// TIA Portal project "plc-programs_V19_S7-1500_PLCSIM_advanced" (V19)
// Vorlageprojekt für das Buch mit Zielsystem S7-1200

(* hardware
DEVICE "S7-1500/ET200MP station_1"  S7-1500 station
   slot 0: "Rail_0"  Rack  6ES7 590-1***0-0AA0
   slot 1: "PLC_1"  CPU 1511-1 PN  6ES7 511-1AK01-0AB0  V2.9
      slot 3: "CPU display_1"  6ES7591-1AA00-0AA0
      slot 32768: "PROFINET interface_1"  X1
         slot 32769: "Port_1"  X1 P1
         slot 32770: "Port_2"  X1 P2
      slot 34817: "Virtual CP interface port_1"  Virtual CP interface port  Virtual CP interface port
*)

// ===== PLC "PLC_1"  CPU 1511-1 PN =====

VAR_GLOBAL   // PLC tag table "Default tag table"
   "Tag_11" AT %M2.4 : Bool;
   "Tag_12" AT %M3.1 : Bool;
END_VAR

VAR_GLOBAL   // PLC tag table "Tag table_Stations123"
   "DI_S1_DiffEntry" AT %I0.2 : Bool;   // S1 item present at infeed
   "DI_S1_VisColor" AT %I0.3 : Bool;   // S1 color/vision detection (blue)
   "DI_S1_PusherBack" AT %I0.4 : Bool;   // S1 pusher fully retracted (home)
   "DI_S1_PusherFront" AT %I0.5 : Bool;   // S1 pusher fully extended
   "DO_S1_Belt2m_A" AT %Q0.1 : Bool;   // S1 short belt A (infeed segment)
   "DO_S2_Belt2m_B" AT %Q0.2 : Bool;   // S2 short belt B (next segment)
   "DO_S1_Belt4m" AT %Q0.3 : Bool;   // S1 long belt past the vision sensor
   "DO_S1_Emitter" AT %Q0.4 : Bool;   // S1 raw material emitter
   "DO_S1_Remover" AT %Q0.5 : Bool;   // S1 rejected blue lid remover
   "DO_S1_Pusher" AT %Q0.6 : Bool;   // S1 pusher extend coil
   "DI_S2_DiffStop0" AT %I0.6 : Bool;   // S2 part present at stop blade 0
   "DI_S2_DiffEntry" AT %I0.7 : Bool;   // S2 part entering station 2
   "r_S2_ArmZpos" AT %ID30 : Real;   // S2 Two-Axis Pick & Place Z axis feedback
   "r_S2_ArmXpos" AT %ID34 : Real;   // S2 Two-Axis Pick & Place X axis feedback
   "DI_S2_ArmRotating" AT %I1.4 : Bool;   // S2 gripper currently rotating
   "DO_S2_Emitter" AT %Q0.7 : Bool;   // S2 base emitter
   "DO_S2_Belt2m_C" AT %Q1.0 : Bool;   // S2 belt carrying parts into the station
   "r_S2_CmdMoveZ" AT %QD30 : Real;   // S2 setpoint for Z axis
   "r_S2_CmdMoveX" AT %QD34 : Real;   // S2 setpoint for X axis
   "DO_S2_Grabe" AT %Q1.2 : Bool;   // S2 gripper close coil
   "DO_S2_RotateRight" AT %Q1.3 : Bool;   // S2 rotate gripper clockwise
   "DO_S2_RotateLeft" AT %Q1.4 : Bool;   // S2 rotate gripper counter-clockwise
   "DO_S2_StopBlade0" AT %Q1.5 : Bool;   // S2 stop blade 0 (near entry)
   "DO_S2_StopBlade1" AT %Q1.6 : Bool;   // S2 stop blade 1 (near assembly)
   "DI_S3_DiffEntry" AT %I1.0 : Bool;   // S3 item entering roller conveyor
   "DI_S3_EntryPart" AT %I1.5 : Bool;   // S3 fingerprint/part present at entry
   "DI_S3_PusherLimit" AT %I1.6 : Bool;   // S3 pusher reached its limit
   "DI_S3_Clamped" AT %I1.7 : Bool;   // S3 clamp closed sensor
   "DI_S3_PalletEntry" AT %I2.0 : Bool;   // S3 empty pallet arrived at loading position
   "DI_S3_PalletLoaded" AT %I2.1 : Bool;   // S3 pallet loaded with a row of items
   "DI_S3_PlateLimit" AT %I2.2 : Bool;   // S3 plate reached its travel limit
   "DI_S3_ElevatorMoving" AT %I2.3 : Bool;   // S3 elevator in motion
   "DO_S3_Clamp" AT %Q2.1 : Bool;   // S3 clamp open/close command
   "DO_S3_OpenPlate" AT %Q2.2 : Bool;   // S3 release plate command
   "DO_S3_PalletLoad" AT %Q2.3 : Bool;   // S3 start loading the pallet
   "DO_S3_Emitter" AT %Q3.2 : Bool;   // S3 Pallet emitter
   "DO_S3_Roller4m_A" AT %Q2.5 : Bool;   // S3 roller conveyor segment A (infeed)
   "DO_S3_Roller4m_B" AT %Q2.6 : Bool;   // S3 roller conveyor segment B (outfeed)
   "DO_S3_ElevatorUp" AT %Q2.7 : Bool;   // S3 raise elevator
   "DO_S3_ElevatorDown" AT %Q3.0 : Bool;   // S3 lower elevator
   "DO_S3_MoveToLimit" AT %Q3.1 : Bool;   // S3 drive elevator to its limit
   "DI_S2_DiffStop1" AT %I1.1 : Bool;   // S2 part present at stop blade 1
   "DI_S2_DiffArmHome" AT %I1.2 : Bool;   // S2 Two-Axis Pick & Place at home
   "DI_S2_ItemDetected" AT %I1.3 : Bool;   // S2 assembly station sees the item
   "DO_S2_Belt2m_D" AT %Q1.1 : Bool;   // S2 outfeed belt after assembly
   "DO_S3_PalletizerBelt" AT %Q1.7 : Bool;   // S3 palletizer transport belt
   "DO_S3_Push" AT %Q2.0 : Bool;   // S3 item pusher (into elevator)
   "DI_S3_PalletExit" AT %I2.4 : Bool;   // S3 finished pallet at exit sensor
   "DO_S3_Remover" AT %Q3.3 : Bool;   // S3 finished-pallet remover
END_VAR

VAR_GLOBAL   // PLC tag table "Tag table_ControlPanel"
   "EStop" AT %I2.5 : Bool;
   "Btn_EstopReset" AT %I2.6 : Bool;
   "Start_Btn" AT %I2.7 : Bool;
   "Stop_Bnt" AT %I3.0 : Bool;
   "AutoMode_S1" AT %I3.1 : Bool;
   "ManualMode_S1" AT %I3.2 : Bool;
   "Lamp_Auto" AT %Q3.4 : Bool;
   "Lamp_Fault" AT %Q3.5 : Bool;
   "Lamp_Run" AT %Q3.6 : Bool;
   "Btn_Start_active" AT %Q3.7 : Bool;
   "Btn_Stop_active" AT %Q4.0 : Bool;
   "EStopReset_Active" AT %Q4.1 : Bool;
   "Btn_ResetCount" AT %I3.3 : Bool;
   "Final_Product_Count" AT %QD38 : DInt;
   "HMI_Start_Btn" AT %M5.0 : Bool;
   "HMI_Sop_Btn" AT %M5.1 : Bool;
   "HMI_CountReset" AT %M5.2 : Bool;
END_VAR

VAR_GLOBAL   // PLC tag table "Tag_table_KPIs"
   "TotalItemsRejected" AT %QD42 : DInt;   // Total rejected items (from FC2 quality reject)
   "TotalRunTime" AT %QD46 : DInt;   // Total run time in seconds
   "ShiftPlannedTime" AT %MW50 : Int;   // Planned production time in seconds (e.g. 28800 = 8h)
   "IdealRate" AT %QD52 : Real;   // Ideal rate items/sec (e.g. 2.5)
   "ActiveAlarmCount" AT %QW56 : Int;   // Number of active alarms
   "TotalDowntime" AT %QD58 : DInt;   // Total downtime in seconds
   "RejectPulse" AT %M2.0 : Bool;   // One-shot pulse on each reject event
   "ProductionPulse" AT %M2.1 : Bool;   // One-shot pulse on each produced item
   "RunTimeEnable" AT %M2.2 : Bool;   // TRUE while line is running (for TON)
   "DowntimeEnable" AT %M2.3 : Bool;   // TRUE while line is stopped (for TON)
   "LidsCount" AT %MD20 : DInt;
   "Alarm_EStop" AT %M4.0 : Bool;
   "Alarm_Fault" AT %M4.1 : Bool;
   "Alarm_LowProduction" AT %M4.2 : Bool;
   "Alarm_HighSort" AT %M4.3 : Bool;
   "Alarm_S2_GripperFault" AT %M4.4 : Bool;
END_VAR

VAR_GLOBAL   // PLC tag table "Standard-Variablentabelle"
   "Tag_1" AT %Q0.0 : Bool;   // Indicates initial communication setup cycle is complete
   "Tag_2" AT %I0.0 : Bool;   // Factory I/O communication link health bit
   "Tag_3" AT %I0.1 : Bool;   // Controls data driver execution for Factory I/O I/O mapping
   "b_S1_PusherReq" AT %M0.0 : Bool;   // S1 pusher request latch
   "Cnt_S3_ItemsInRow" AT %MW20 : Int;   // S3 count of items in current row (CTU counter_0 CV)
   "b_S3_Trig_ElevatorStop" AT %M0.2 : Bool;   // N_TRIG on ElevatorMoving
   "b_S3_Trig_Clamp" AT %M0.3 : Bool;   // N_TRIG on Push for clamp sequence
   "b_S3_Trig_PalletLoaded" AT %M0.4 : Bool;   // P_TRIG on PalletLoaded for elevator-up
   "b_S3_Trig_RowStart" AT %M0.5 : Bool;   // N_TRIG on Push for counter_1 step
   "b_S3_Flg_ElevatorClear" AT %M0.6 : Bool;   // condition for counter_2 step
   "b_S3_Flg_ArmAtTop" AT %M0.7 : Bool;   // condition for counter_1 step
   "b_S3_Flg_RowReady" AT %M1.0 : Bool;   // condition to clear Pallet Load
   "b_S3_Trig_OpenPlate" AT %M1.1 : Bool;   // N_TRIG on ElevatorDown for plate open
   "b_S3_Trig_PlateCycle" AT %M1.2 : Bool;   // N_TRIG on Push for plate cycle
   "Tag_4" AT %M1.3 : Bool;
   "Tag_5" AT %M1.4 : Bool;
   "Tag_6" AT %M1.5 : Bool;
   "Tag_7" AT %M1.6 : Bool;
   "Tag_8" AT %MW30 : Int;
   "Tag_9" AT %M1.7 : Bool;
   "Tag_10" AT %M3.0 : Bool;
END_VAR

DATA_BLOCK "DB_ControlPanel"   // DB7
{ S7_Optimized_Access := 'TRUE' }
VERSION : 0.1
   VAR
      EStopActive : Bool;
      LineEnable : Bool;
      StartReq : Bool;
      StopReq : Bool;
      AutoMode : Bool;
      ManualMode : Bool;
      LineRunning : Bool;
      LampRun : Bool;
      LampFault : Bool;
      LampAuto : Bool;
   END_VAR
BEGIN
END_DATA_BLOCK

DATA_BLOCK "DB50_KPIs"   // DB9
{ S7_Optimized_Access := 'TRUE' }
VERSION : 0.1
   VAR
      ProductionCount : DInt;   // Total items produced
      LoadedPalletCount : Int;   // Total finished pallets at exit
      SortedCount : DInt;   // Number of blue lids sorted out
      SortRate : Real;   // sort percentage
      CycleTime : Real;   // Time between two consecutive items (ms)
      Throughput : Real;   // Items per minute
      Availability : Real;   // Run time ÷ Planned time × 100
      Performance : Real;   // Actual rate ÷ Ideal rate × 100
      Yield : Real;   // (total - sorted) / total
      OEE : Real;   // Count of active alarms
      ActiveAlarms : Int;   // Count of active alarms
      Downtime : DInt;   // Total downtime in seconds
      Status : Word;   // 0=OK, 1=Fault, 2=ESTOP
      Timestamp : DTL;   // Current PLC time
   END_VAR
BEGIN
END_DATA_BLOCK

DATA_BLOCK "KPIs_DB"   // DB14
{ S7_Optimized_Access := 'TRUE' }
VERSION : 0.1
// stored: InstanceOfName KPIs
"KPIs"
BEGIN
END_DATA_BLOCK

// folder: System blocks/Program resources

DATA_BLOCK "IEC_Timer_0_DB"   // DB1
{ S7_Optimized_Access := 'TRUE' }
AUTHOR : Simatic
FAMILY : IEC
NAME : IEC_TMR
VERSION : 1.0
// stored: InstanceOfName IEC_TIMER
"IEC_TIMER"
BEGIN
END_DATA_BLOCK

DATA_BLOCK "counter_2"   // DB2
{ S7_Optimized_Access := 'TRUE' }
AUTHOR : Simatic
FAMILY : IEC
NAME : CNTR
VERSION : 1.0
// stored: InstanceOfName IEC_COUNTER
"IEC_COUNTER"
BEGIN
END_DATA_BLOCK

DATA_BLOCK "Counter_0"   // DB3
{ S7_Optimized_Access := 'TRUE' }
AUTHOR : Simatic
FAMILY : IEC
NAME : CNTR
VERSION : 1.0
// stored: InstanceOfName IEC_COUNTER
"IEC_COUNTER"
BEGIN
END_DATA_BLOCK

DATA_BLOCK "Timer_1"   // DB4
{ S7_Optimized_Access := 'TRUE' }
AUTHOR : Simatic
FAMILY : IEC
NAME : IEC_TMR
VERSION : 1.0
// stored: InstanceOfName IEC_TIMER
"IEC_TIMER"
BEGIN
END_DATA_BLOCK

DATA_BLOCK "counter_1"   // DB5
{ S7_Optimized_Access := 'TRUE' }
AUTHOR : Simatic
FAMILY : IEC
NAME : CNTR
VERSION : 1.0
// stored: InstanceOfName IEC_COUNTER
"IEC_COUNTER"
BEGIN
END_DATA_BLOCK

DATA_BLOCK "Counter_3"   // DB6
{ S7_Optimized_Access := 'TRUE' }
AUTHOR : Simatic
FAMILY : IEC
NAME : CNTR
VERSION : 1.0
// stored: InstanceOfName IEC_COUNTER
"IEC_COUNTER"
BEGIN
END_DATA_BLOCK

DATA_BLOCK "Counter_4"   // DB8
{ S7_Optimized_Access := 'TRUE' }
AUTHOR : Simatic
FAMILY : IEC
NAME : CNTR
VERSION : 1.0
// stored: InstanceOfName IEC_COUNTER
"IEC_COUNTER"
BEGIN
END_DATA_BLOCK

DATA_BLOCK "Ton_TotalRunTime"   // DB10
{ S7_Optimized_Access := 'TRUE' }
AUTHOR : Simatic
FAMILY : IEC
NAME : IEC_TMR
VERSION : 1.0
// stored: InstanceOfName IEC_TIMER
"IEC_TIMER"
BEGIN
END_DATA_BLOCK

DATA_BLOCK "Ton_TotalDowntime"   // DB11
{ S7_Optimized_Access := 'TRUE' }
AUTHOR : Simatic
FAMILY : IEC
NAME : IEC_TMR
VERSION : 1.0
// stored: InstanceOfName IEC_TIMER
"IEC_TIMER"
BEGIN
END_DATA_BLOCK

DATA_BLOCK "Cnt_TotalRejected"   // DB12
{ S7_Optimized_Access := 'TRUE' }
AUTHOR : Simatic
FAMILY : IEC
NAME : CNTR
VERSION : 1.0
// stored: InstanceOfName IEC_COUNTER
"IEC_COUNTER"
BEGIN
END_DATA_BLOCK

DATA_BLOCK "FP_Counter"   // DB15
{ S7_Optimized_Access := 'TRUE' }
AUTHOR : Simatic
FAMILY : IEC
NAME : CNTR
VERSION : 1.0
// stored: InstanceOfName IEC_COUNTER
"IEC_COUNTER"
BEGIN
END_DATA_BLOCK

DATA_BLOCK "Step5_counter"   // DB16
{ S7_Optimized_Access := 'TRUE' }
AUTHOR : Simatic
FAMILY : IEC
NAME : CNTR
VERSION : 1.0
// stored: InstanceOfName IEC_COUNTER
"IEC_COUNTER"
BEGIN
END_DATA_BLOCK

DATA_BLOCK "Cnt_greenlids"   // DB17
{ S7_Optimized_Access := 'TRUE' }
AUTHOR : Simatic
FAMILY : IEC
NAME : CNTR
VERSION : 1.0
// stored: InstanceOfName IEC_COUNTER
"IEC_COUNTER"
BEGIN
END_DATA_BLOCK

// folder: (top level)

FUNCTION_BLOCK "KPIs"   // FB1, SCL
{ S7_Optimized_Access := 'TRUE' }
VERSION : 0.1
   VAR_INPUT
      CycleCount : DInt;
      SortedCount : DInt;
      RunTime : DInt;
      PlannedTime : DInt;
      Downtime : DInt;
      IdealRate : Real;
      EStop : Bool;
   END_VAR
   VAR_IN_OUT
      ActiveAlarmCount : Int;
   END_VAR
   VAR
      LastCycleCount : DInt;
      LastItemTime : DTL;
   END_VAR
   VAR_TEMP
      CurrentTime : DTL;
      RetVal : Int;
   END_VAR
BEGIN
   // Read current system time into our Temp variable
   #RetVal := RD_SYS_T(#CurrentTime);
   "DB50_KPIs".Timestamp := #CurrentTime;

   "DB50_KPIs".ProductionCount := #CycleCount;
   "DB50_KPIs".SortedCount := #SortedCount;

   // Quality and Reject Rate
   IF "LidsCount" > 0 THEN
       "DB50_KPIs".SortRate := 100.0 * DINT_TO_REAL(#SortedCount) / DINT_TO_REAL("LidsCount"+#SortedCount);
       "DB50_KPIs".Yield := 100.0 * DINT_TO_REAL("LidsCount") / DINT_TO_REAL("LidsCount"+#SortedCount);
   END_IF;

   // Cycle Time (using T_DIFF for S7-1200 compatibility)
   IF #CycleCount > #LastCycleCount THEN
       IF #LastCycleCount > 0 THEN // Prevent massive time calculation on the very first part
           "DB50_KPIs".CycleTime := DINT_TO_REAL(TIME_TO_DINT(T_DIFF(IN1 := #CurrentTime, IN2 := #LastItemTime)));
       END_IF;
       #LastItemTime := #CurrentTime;
       #LastCycleCount := #CycleCount;
   END_IF;

   // Throughput & Performance
   IF "DB50_KPIs".CycleTime > 0.0 THEN
       "DB50_KPIs".Throughput := 60000.0 / "DB50_KPIs".CycleTime; // Calculates Parts Per Minute

       IF #IdealRate > 0.0 THEN
           // Use Throughput directly to ensure both are in Parts Per Minute
           "DB50_KPIs".Performance := 100.0 * ("DB50_KPIs".Throughput / #IdealRate);
       END_IF;
   END_IF;

   // Availability & OEE
   IF #PlannedTime > 0 THEN
       // Divide RunTime by 1000.0 to convert milliseconds to seconds
       "DB50_KPIs".Availability := 100.0 * (DINT_TO_REAL(#RunTime) / 1000.0) / DINT_TO_REAL(#PlannedTime);
   END_IF;
   "DB50_KPIs".OEE := ("DB50_KPIs".Availability * "DB50_KPIs".Performance * "DB50_KPIs".Yield) / 10000.0;

   // Status
   IF NOT #EStop THEN
       "DB50_KPIs".Status := 2;
   ELSIF #ActiveAlarmCount > 0 THEN
       "DB50_KPIs".Status := 1;
   ELSE
       "DB50_KPIs".Status := 0;
   END_IF;

   "DB50_KPIs".ActiveAlarms := #ActiveAlarmCount;
   "DB50_KPIs".Downtime := #Downtime;

   // --- Active alarm count ---
   #ActiveAlarmCount := 0;
   IF "Alarm_EStop" THEN
       #ActiveAlarmCount := #ActiveAlarmCount + 1;
   END_IF;
   IF "Alarm_Fault" THEN
       #ActiveAlarmCount := #ActiveAlarmCount + 1;
   END_IF;
   IF "Alarm_LowProduction" THEN
       #ActiveAlarmCount := #ActiveAlarmCount + 1;
   END_IF;
   IF "Alarm_HighSort" THEN
       #ActiveAlarmCount := #ActiveAlarmCount + 1;
   END_IF;

   IF "Alarm_S2_GripperFault" THEN
       #ActiveAlarmCount := #ActiveAlarmCount + 1;
   END_IF;
END_FUNCTION_BLOCK

FUNCTION "Station1" : Void   // FC1, LAD
TITLE = Infeed & Color Sorting
{ S7_Optimized_Access := 'TRUE' }
AUTHOR : Youness Tebbaq
VERSION : 0.1
// "Station 1 (Infeed & Color Sorting). The emitter spawns (Blue/Green) lids onto the main conveyor. A diffuse sensor starts the 4 m belt only when the 2 m belts are free (anti-jam). The vision sensor triggers a pusher request whene a blue lid detected; a short timer then fires the pusher. When the pusher reaches its front limit it retracts and the request flag is cleared. The station runs	
// in a continuous loop with no start/stop logic."
BEGIN

REGION Network 1: Always run — Emitter and Remover
   // Emitter and Remover are permanently ON. The emitter continuously
   // spawns Blue/Green lids  into the line; the remover continuously deletes
   // Blue lids at the end of the diverted lane .
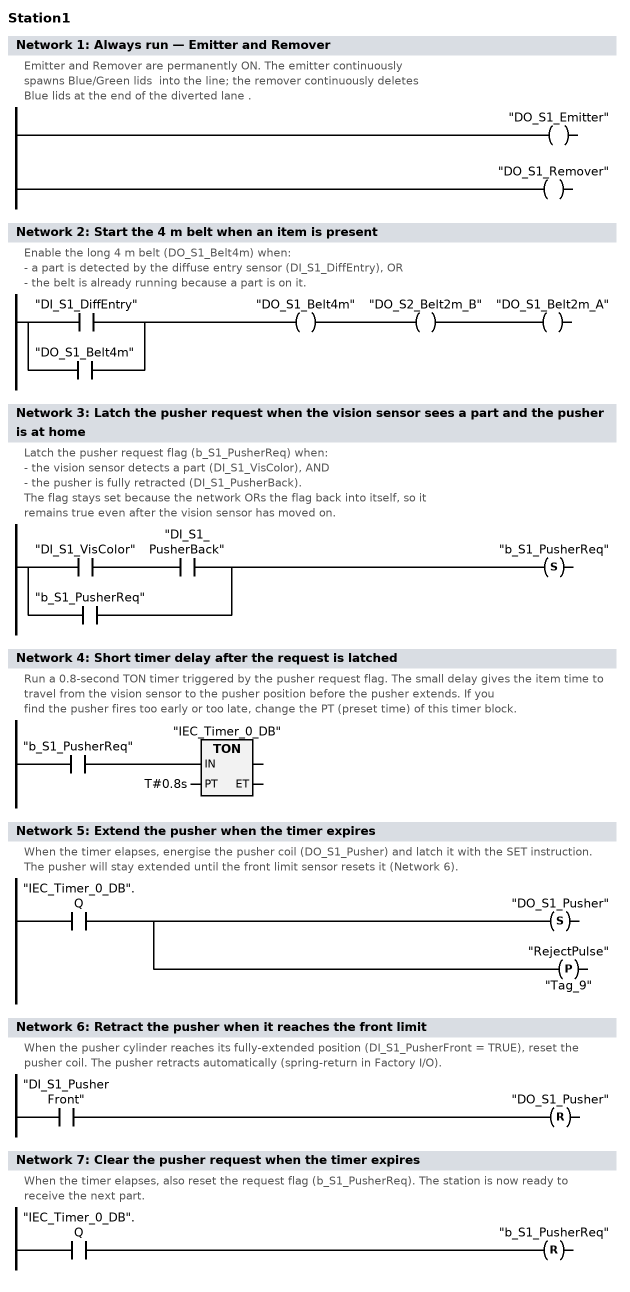
   RUNG wire#powerrail
      Coil( "DO_S1_Emitter" )
   END_RUNG
   RUNG wire#powerrail
      Coil( "DO_S1_Remover" )
   END_RUNG
   // the same network as SCL:
   "DO_S1_Emitter" := TRUE;
   "DO_S1_Remover" := TRUE;
END_REGION

REGION Network 2: Start the 4 m belt when an item is present
   // Enable the long 4 m belt (DO_S1_Belt4m) when:
   //   - a part is detected by the diffuse entry sensor (DI_S1_DiffEntry), OR
   //   - the belt is already running because a part is on it.
   RUNG wire#powerrail
      Contact( "DI_S1_DiffEntry" )
      wire#w1
      Coil( "DO_S1_Belt4m" )
      Coil( "DO_S2_Belt2m_B" )
      Coil( "DO_S1_Belt2m_A" )
   END_RUNG
   RUNG wire#powerrail
      Contact( "DO_S1_Belt4m" )
   END_RUNG wire#w1
   // the same network as SCL:
   "DO_S1_Belt4m" := "DI_S1_DiffEntry" OR "DO_S1_Belt4m";
   "DO_S2_Belt2m_B" := "DO_S1_Belt4m";
   "DO_S1_Belt2m_A" := "DO_S1_Belt4m";
END_REGION

REGION Network 3: Latch the pusher request when the vision sensor sees a part and the pusher is at home
   // Latch the pusher request flag (b_S1_PusherReq) when:
   //   - the vision sensor detects a part (DI_S1_VisColor), AND
   //   - the pusher is fully retracted (DI_S1_PusherBack).
   // The flag stays set because the network ORs the flag back into itself, so it
   // remains true even after the vision sensor has moved on.
   RUNG wire#powerrail
      Contact( "DI_S1_VisColor" )
      Contact( "DI_S1_PusherBack" )
      wire#w1
      S_Coil( "b_S1_PusherReq" )
   END_RUNG
   RUNG wire#powerrail
      Contact( "b_S1_PusherReq" )
   END_RUNG wire#w1
   // the same network as SCL:
   IF ("DI_S1_VisColor" AND "DI_S1_PusherBack") OR "b_S1_PusherReq" THEN "b_S1_PusherReq" := TRUE; END_IF;
END_REGION

REGION Network 4: Short timer delay after the request is latched
   // Run a 0.8-second TON timer triggered by the pusher request flag. The small delay gives the item time to travel from the vision sensor to the pusher position before the pusher extends. If you
   // find the pusher fires too early or too late, change the PT (preset time) of this timer block.
   "IEC_Timer_0_DB".TON(IN := "b_S1_PusherReq", PT := T#0.8s);
END_REGION

REGION Network 5: Extend the pusher when the timer expires
   // When the timer elapses, energise the pusher coil (DO_S1_Pusher) and latch it with the SET instruction. The pusher will stay extended until the front limit sensor resets it (Network 6).
   IF "IEC_Timer_0_DB".Q THEN "DO_S1_Pusher" := TRUE; END_IF;
   "RejectPulse" := "IEC_Timer_0_DB".Q AND NOT "Tag_9";   // rising edge
   "Tag_9" := "IEC_Timer_0_DB".Q;
END_REGION

REGION Network 6: Retract the pusher when it reaches the front limit
   // When the pusher cylinder reaches its fully-extended position (DI_S1_PusherFront = TRUE), reset the pusher coil. The pusher retracts automatically (spring-return in Factory I/O).
   RUNG wire#powerrail
      Contact( "DI_S1_PusherFront" )
      R_Coil( "DO_S1_Pusher" )
   END_RUNG
   // the same network as SCL:
   IF "DI_S1_PusherFront" THEN "DO_S1_Pusher" := FALSE; END_IF;
END_REGION

REGION Network 7: Clear the pusher request when the timer expires
   // When the timer elapses, also reset the request flag (b_S1_PusherReq). The station is now ready to receive the next part.
   RUNG wire#powerrail
      Contact( "IEC_Timer_0_DB".Q )
      R_Coil( "b_S1_PusherReq" )
   END_RUNG
   // the same network as SCL:
   IF "IEC_Timer_0_DB".Q THEN "b_S1_PusherReq" := FALSE; END_IF;
END_REGION
END_FUNCTION

FUNCTION "Station2" : Void   // FC2, LAD
TITLE = Station 2 — Assembly
{ S7_Optimized_Access := 'TRUE' }
AUTHOR : Youness Tebbaq
VERSION : 0.1
// Station 2 (Assembly). 
// -The Two-Axis Pick & Place assembles a Product Lid onto a Product Base. 
// -A diffuse sensor at the entry (DI_S2_DiffEntry) starts belt C (DO_S2_Belt2m_C); once the part is in position the stop blade (DO_S2_StopBlade0) holds it.
// -The arm executes a fixed pick-and-place sequence by driving the Z axis first (r_S2_CmdMoveZ = 10.0 to lower, 0.0 to raise), then the X axis (r_S2_CmdMoveX = 10.0 to move over the base, 0.0 to return).
// -The gripper is closed (DO_S2_Grabe) while the arm is above the base.
// - Rotation (DO_S2_RotateRight / DO_S2_RotateLeft) is used to place the lid with the correct orientation. 
// -The cycle ends when the arm returns to the home sensor (DI_S2_DiffArmHome).
   VAR_TEMP   // added for the SCL form of the ladder/FBD networks
      _w1 : Bool;
   END_VAR
BEGIN

REGION Network 1: Start belt C and latch the emitter when an item is present
   // Latch the emitter (DO_S2_Emitter) when a part enters station 2 (DI_S2_DiffEntry). The emitter stays ON because the network ORs the latched output back into itself. The emitter is cleared in Network 4 by the stop blade 1 sensor.
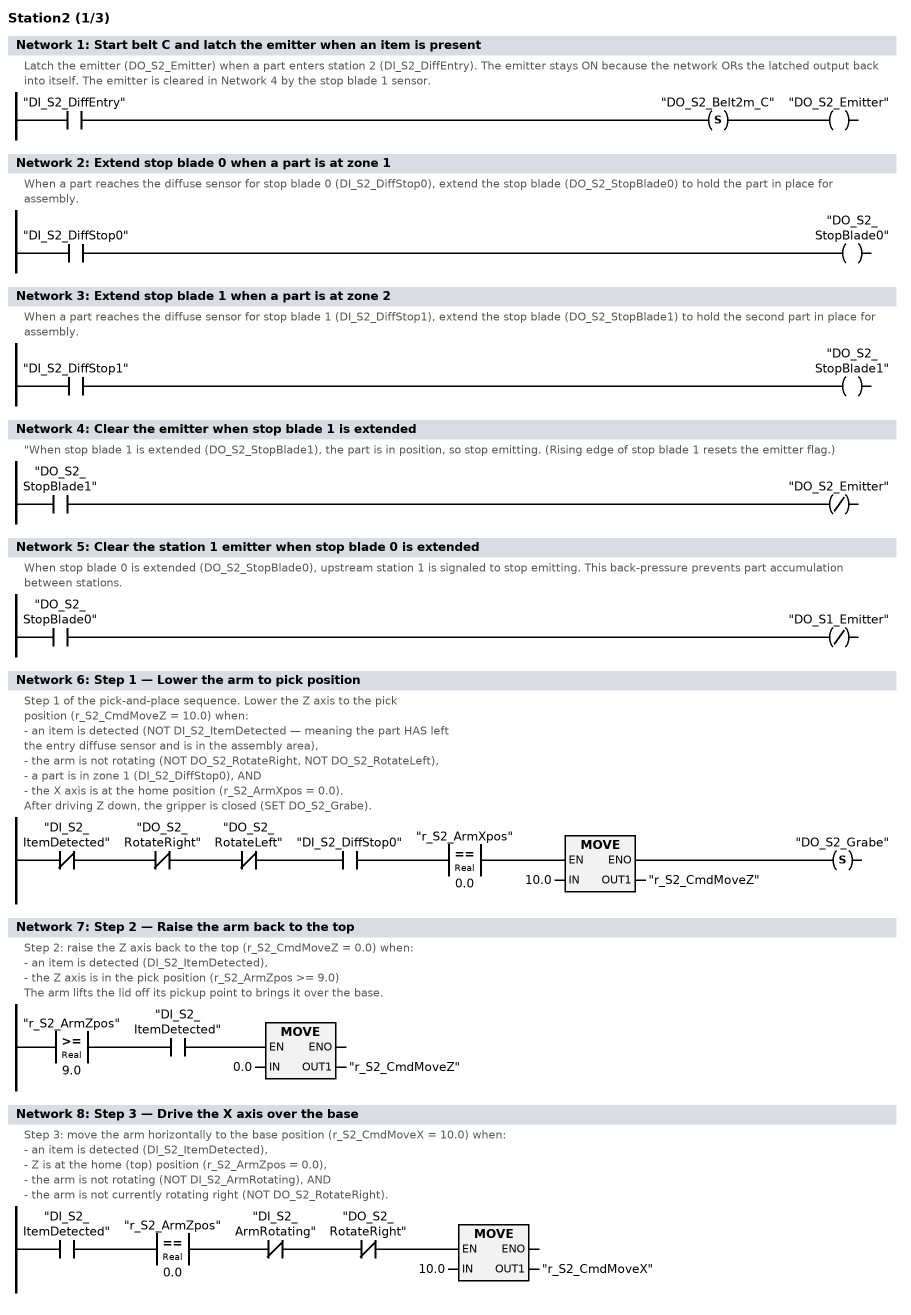
   RUNG wire#powerrail
      Contact( "DI_S2_DiffEntry" )
      S_Coil( "DO_S2_Belt2m_C" )
      Coil( "DO_S2_Emitter" )
   END_RUNG
   // the same network as SCL:
   IF "DI_S2_DiffEntry" THEN "DO_S2_Belt2m_C" := TRUE; END_IF;
   "DO_S2_Emitter" := "DI_S2_DiffEntry";
END_REGION

REGION Network 2: Extend stop blade 0 when a part is at zone 1
   // When a part reaches the diffuse sensor for stop blade 0 (DI_S2_DiffStop0), extend the stop blade (DO_S2_StopBlade0) to hold the part in place for assembly.
   RUNG wire#powerrail
      Contact( "DI_S2_DiffStop0" )
      Coil( "DO_S2_StopBlade0" )
   END_RUNG
   // the same network as SCL:
   "DO_S2_StopBlade0" := "DI_S2_DiffStop0";
END_REGION

REGION Network 3: Extend stop blade 1 when a part is at zone 2
   // When a part reaches the diffuse sensor for stop blade 1 (DI_S2_DiffStop1), extend the stop blade (DO_S2_StopBlade1) to hold the second part in place for assembly.
   RUNG wire#powerrail
      Contact( "DI_S2_DiffStop1" )
      Coil( "DO_S2_StopBlade1" )
   END_RUNG
   // the same network as SCL:
   "DO_S2_StopBlade1" := "DI_S2_DiffStop1";
END_REGION

REGION Network 4: Clear the emitter when stop blade 1 is extended
   // "When stop blade 1 is extended (DO_S2_StopBlade1), the part is in position, so stop emitting. (Rising edge of stop blade 1 resets the emitter flag.)
   RUNG wire#powerrail
      Contact( "DO_S2_StopBlade1" )
      I_Coil( "DO_S2_Emitter" )
   END_RUNG
   // the same network as SCL:
   "DO_S2_Emitter" := NOT "DO_S2_StopBlade1";
END_REGION

REGION Network 5: Clear the station 1 emitter when stop blade 0 is extended
   // When stop blade 0 is extended (DO_S2_StopBlade0), upstream station 1 is signaled to stop emitting. This back-pressure prevents part accumulation between stations.
   RUNG wire#powerrail
      Contact( "DO_S2_StopBlade0" )
      I_Coil( "DO_S1_Emitter" )
   END_RUNG
   // the same network as SCL:
   "DO_S1_Emitter" := NOT "DO_S2_StopBlade0";
END_REGION

REGION Network 6: Step 1 — Lower the arm to pick position
   // Step 1 of the pick-and-place sequence. Lower the Z axis to the pick
   // position (r_S2_CmdMoveZ = 10.0) when:
   //   - an item is detected (NOT DI_S2_ItemDetected — meaning the part HAS left
   //     the entry diffuse sensor and is in the assembly area),
   //   - the arm is not rotating (NOT DO_S2_RotateRight, NOT DO_S2_RotateLeft),
   //   - a part is in zone 1 (DI_S2_DiffStop0), AND
   //   - the X axis is at the home position (r_S2_ArmXpos = 0.0).
   // After driving Z down, the gripper is closed (SET DO_S2_Grabe).
   RUNG wire#powerrail
      I_Contact( "DI_S2_ItemDetected" )
      I_Contact( "DO_S2_RotateRight" )
      I_Contact( "DO_S2_RotateLeft" )
      Contact( "DI_S2_DiffStop0" )
      { S7_Templates := "SrcType := Real" } EQ_Contact(in1 := "r_S2_ArmXpos", in2 := 0.0)
      Move(in := 10.0, out1 => "r_S2_CmdMoveZ")
      S_Coil( "DO_S2_Grabe" )
   END_RUNG
   // the same network as SCL:
   IF NOT "DI_S2_ItemDetected" AND NOT "DO_S2_RotateRight" AND NOT "DO_S2_RotateLeft" AND "DI_S2_DiffStop0" AND ("r_S2_ArmXpos" = 0.0) THEN
       "r_S2_CmdMoveZ" := 10.0;
       "DO_S2_Grabe" := TRUE;
   END_IF;
END_REGION

REGION Network 7: Step 2 — Raise the arm back to the top
   // Step 2: raise the Z axis back to the top (r_S2_CmdMoveZ = 0.0) when:
   //   - an item is detected (DI_S2_ItemDetected),
   //   - the Z axis is in the pick position (r_S2_ArmZpos >= 9.0)
   // The arm lifts the lid off its pickup point to brings it over the base.
   RUNG wire#powerrail
      { S7_Templates := "SrcType := Real" } GE_Contact(in1 := "r_S2_ArmZpos", in2 := 9.0)
      Contact( "DI_S2_ItemDetected" )
      Move(in := 0.0, out1 => "r_S2_CmdMoveZ")
   END_RUNG
   // the same network as SCL:
   IF ("r_S2_ArmZpos" >= 9.0) AND "DI_S2_ItemDetected" THEN "r_S2_CmdMoveZ" := 0.0; END_IF;
END_REGION

REGION Network 8: Step 3 — Drive the X axis over the base
   // Step 3: move the arm horizontally to the base position (r_S2_CmdMoveX = 10.0) when:
   //   - an item is detected (DI_S2_ItemDetected),
   //   - Z is at the home (top) position (r_S2_ArmZpos = 0.0),
   //    - the arm is not rotating (NOT DI_S2_ArmRotating), AND
   //   - the arm is not currently rotating right (NOT DO_S2_RotateRight).
   RUNG wire#powerrail
      Contact( "DI_S2_ItemDetected" )
      { S7_Templates := "SrcType := Real" } EQ_Contact(in1 := "r_S2_ArmZpos", in2 := 0.0)
      I_Contact( "DI_S2_ArmRotating" )
      I_Contact( "DO_S2_RotateRight" )
      Move(in := 10.0, out1 => "r_S2_CmdMoveX")
   END_RUNG
   // the same network as SCL:
   IF "DI_S2_ItemDetected" AND ("r_S2_ArmZpos" = 0.0) AND NOT "DI_S2_ArmRotating" AND NOT "DO_S2_RotateRight" THEN
       "r_S2_CmdMoveX" := 10.0;
   END_IF;
END_REGION

REGION Network 9: Step 4 — Lower the arm onto the base
   // Step 4: lower the Z axis onto the base position
   // (r_S2_CmdMoveZ = 10.0) when:
   //   - an item is detected (DI_S2_ItemDetected),
   //   - stop blade 1 is set (DI_S2_DiffStop1),
   //   - the X axis has reached the base position (r_S2_ArmXpos >= 9.0), AND
   //   - Z is at the home (top) position (r_S2_ArmZpos = 0.0).
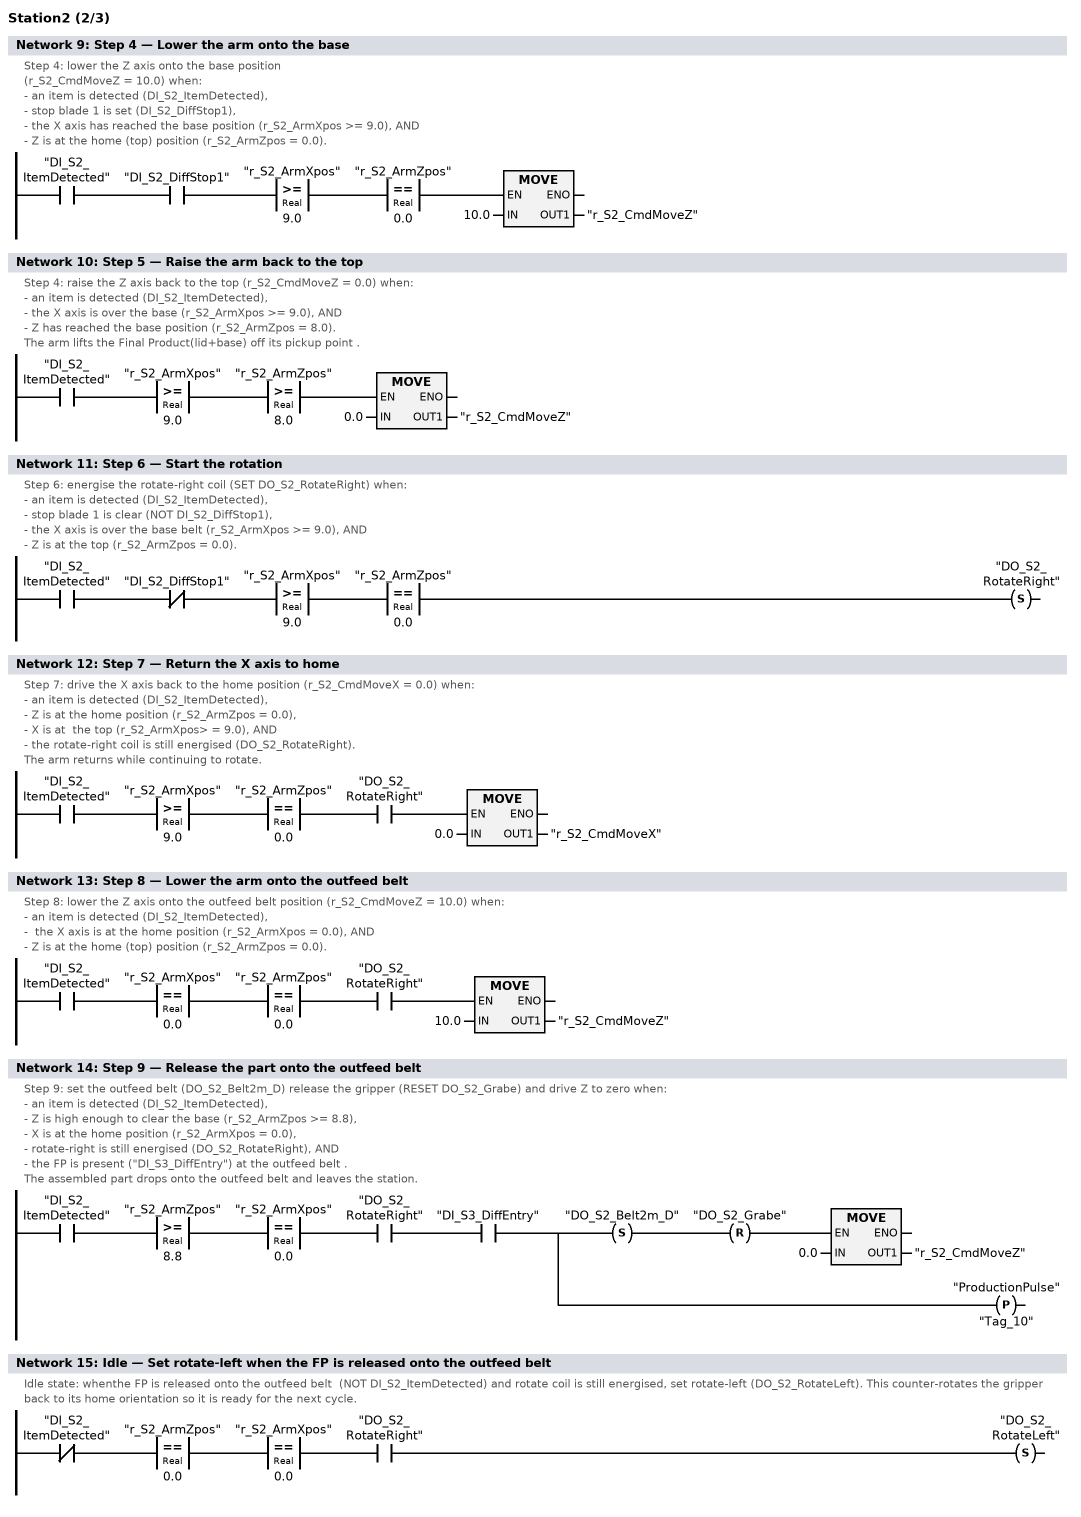
   RUNG wire#powerrail
      Contact( "DI_S2_ItemDetected" )
      Contact( "DI_S2_DiffStop1" )
      { S7_Templates := "SrcType := Real" } GE_Contact(in1 := "r_S2_ArmXpos", in2 := 9.0)
      { S7_Templates := "SrcType := Real" } EQ_Contact(in1 := "r_S2_ArmZpos", in2 := 0.0)
      Move(in := 10.0, out1 => "r_S2_CmdMoveZ")
   END_RUNG
   // the same network as SCL:
   IF "DI_S2_ItemDetected" AND "DI_S2_DiffStop1" AND ("r_S2_ArmXpos" >= 9.0) AND ("r_S2_ArmZpos" = 0.0) THEN
       "r_S2_CmdMoveZ" := 10.0;
   END_IF;
END_REGION

REGION Network 10: Step 5 — Raise the arm back to the top
   // Step 4: raise the Z axis back to the top (r_S2_CmdMoveZ = 0.0) when:
   //   - an item is detected (DI_S2_ItemDetected),
   //   - the X axis is over the base (r_S2_ArmXpos >= 9.0), AND
   //   - Z has reached the base position (r_S2_ArmZpos = 8.0).
   // The arm lifts the Final Product(lid+base) off its pickup point .
   RUNG wire#powerrail
      Contact( "DI_S2_ItemDetected" )
      { S7_Templates := "SrcType := Real" } GE_Contact(in1 := "r_S2_ArmXpos", in2 := 9.0)
      { S7_Templates := "SrcType := Real" } GE_Contact(in1 := "r_S2_ArmZpos", in2 := 8.0)
      Move(in := 0.0, out1 => "r_S2_CmdMoveZ")
   END_RUNG
   // the same network as SCL:
   IF "DI_S2_ItemDetected" AND ("r_S2_ArmXpos" >= 9.0) AND ("r_S2_ArmZpos" >= 8.0) THEN
       "r_S2_CmdMoveZ" := 0.0;
   END_IF;
END_REGION

REGION Network 11: Step 6 — Start the rotation
   // Step 6: energise the rotate-right coil (SET DO_S2_RotateRight) when:
   //   - an item is detected (DI_S2_ItemDetected),
   //   - stop blade 1 is clear (NOT DI_S2_DiffStop1),
   //   - the X axis is over the base belt (r_S2_ArmXpos >= 9.0), AND
   //   - Z is at the top (r_S2_ArmZpos = 0.0).
   RUNG wire#powerrail
      Contact( "DI_S2_ItemDetected" )
      I_Contact( "DI_S2_DiffStop1" )
      { S7_Templates := "SrcType := Real" } GE_Contact(in1 := "r_S2_ArmXpos", in2 := 9.0)
      { S7_Templates := "SrcType := Real" } EQ_Contact(in1 := "r_S2_ArmZpos", in2 := 0.0)
      S_Coil( "DO_S2_RotateRight" )
   END_RUNG
   // the same network as SCL:
   IF "DI_S2_ItemDetected" AND NOT "DI_S2_DiffStop1" AND ("r_S2_ArmXpos" >= 9.0) AND ("r_S2_ArmZpos" = 0.0) THEN
       "DO_S2_RotateRight" := TRUE;
   END_IF;
END_REGION

REGION Network 12: Step 7 — Return the X axis to home
   // Step 7: drive the X axis back to the home position (r_S2_CmdMoveX = 0.0) when:
   //   - an item is detected (DI_S2_ItemDetected),
   //   - Z is at the home position (r_S2_ArmZpos = 0.0),
   //   - X is at  the top (r_S2_ArmXpos> = 9.0), AND
   //   - the rotate-right coil is still energised (DO_S2_RotateRight).
   // The arm returns while continuing to rotate.
   RUNG wire#powerrail
      Contact( "DI_S2_ItemDetected" )
      { S7_Templates := "SrcType := Real" } GE_Contact(in1 := "r_S2_ArmXpos", in2 := 9.0)
      { S7_Templates := "SrcType := Real" } EQ_Contact(in1 := "r_S2_ArmZpos", in2 := 0.0)
      Contact( "DO_S2_RotateRight" )
      Move(in := 0.0, out1 => "r_S2_CmdMoveX")
   END_RUNG
   // the same network as SCL:
   IF "DI_S2_ItemDetected" AND ("r_S2_ArmXpos" >= 9.0) AND ("r_S2_ArmZpos" = 0.0) AND "DO_S2_RotateRight" THEN
       "r_S2_CmdMoveX" := 0.0;
   END_IF;
END_REGION

REGION Network 13: Step 8 — Lower the arm onto the outfeed belt
   // Step 8: lower the Z axis onto the outfeed belt position (r_S2_CmdMoveZ = 10.0) when:
   //   - an item is detected (DI_S2_ItemDetected),
   //   -  the X axis is at the home position (r_S2_ArmXpos = 0.0), AND
   //   - Z is at the home (top) position (r_S2_ArmZpos = 0.0).
   RUNG wire#powerrail
      Contact( "DI_S2_ItemDetected" )
      { S7_Templates := "SrcType := Real" } EQ_Contact(in1 := "r_S2_ArmXpos", in2 := 0.0)
      { S7_Templates := "SrcType := Real" } EQ_Contact(in1 := "r_S2_ArmZpos", in2 := 0.0)
      Contact( "DO_S2_RotateRight" )
      Move(in := 10.0, out1 => "r_S2_CmdMoveZ")
   END_RUNG
   // the same network as SCL:
   IF "DI_S2_ItemDetected" AND ("r_S2_ArmXpos" = 0.0) AND ("r_S2_ArmZpos" = 0.0) AND "DO_S2_RotateRight" THEN
       "r_S2_CmdMoveZ" := 10.0;
   END_IF;
END_REGION

REGION Network 14: Step 9 — Release the part onto the outfeed belt
   // Step 9: set the outfeed belt (DO_S2_Belt2m_D) release the gripper (RESET DO_S2_Grabe) and drive Z to zero when:
   //   - an item is detected (DI_S2_ItemDetected),
   //   - Z is high enough to clear the base (r_S2_ArmZpos >= 8.8),
   //   - X is at the home position (r_S2_ArmXpos = 0.0),
   //   - rotate-right is still energised (DO_S2_RotateRight), AND
   //   - the FP is present ("DI_S3_DiffEntry") at the outfeed belt .
   // The assembled part drops onto the outfeed belt and leaves the station.
   #_w1 := "DI_S2_ItemDetected" AND ("r_S2_ArmZpos" >= 8.8) AND ("r_S2_ArmXpos" = 0.0) AND "DO_S2_RotateRight" AND "DI_S3_DiffEntry";
   IF #_w1 THEN
       "DO_S2_Belt2m_D" := TRUE;
       "DO_S2_Grabe" := FALSE;
       "r_S2_CmdMoveZ" := 0.0;
   END_IF;
   "ProductionPulse" := #_w1 AND NOT "Tag_10";   // rising edge
   "Tag_10" := #_w1;
END_REGION

REGION Network 15: Idle — Set rotate-left when the FP is released onto the outfeed belt
   // Idle state: whenthe FP is released onto the outfeed belt  (NOT DI_S2_ItemDetected) and rotate coil is still energised, set rotate-left (DO_S2_RotateLeft). This counter-rotates the gripper back to its home orientation so it is ready for the next cycle.
   RUNG wire#powerrail
      I_Contact( "DI_S2_ItemDetected" )
      { S7_Templates := "SrcType := Real" } EQ_Contact(in1 := "r_S2_ArmZpos", in2 := 0.0)
      { S7_Templates := "SrcType := Real" } EQ_Contact(in1 := "r_S2_ArmXpos", in2 := 0.0)
      Contact( "DO_S2_RotateRight" )
      S_Coil( "DO_S2_RotateLeft" )
   END_RUNG
   // the same network as SCL:
   IF NOT "DI_S2_ItemDetected" AND ("r_S2_ArmZpos" = 0.0) AND ("r_S2_ArmXpos" = 0.0) AND "DO_S2_RotateRight" THEN
       "DO_S2_RotateLeft" := TRUE;
   END_IF;
END_REGION

REGION Network 16: Home position — clear both rotation coils
   // When the arm reaches the home sensor (DI_S2_DiffArmHome), Z and X are both at zero, and both rotation coils still energised.
   //  The arm is now in itshome position and ready to start a new cycle.
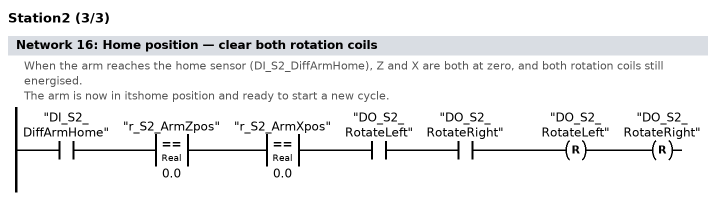
   RUNG wire#powerrail
      Contact( "DI_S2_DiffArmHome" )
      { S7_Templates := "SrcType := Real" } EQ_Contact(in1 := "r_S2_ArmZpos", in2 := 0.0)
      { S7_Templates := "SrcType := Real" } EQ_Contact(in1 := "r_S2_ArmXpos", in2 := 0.0)
      Contact( "DO_S2_RotateLeft" )
      Contact( "DO_S2_RotateRight" )
      R_Coil( "DO_S2_RotateLeft" )
      R_Coil( "DO_S2_RotateRight" )
   END_RUNG
   // the same network as SCL:
   #_w1 := "DI_S2_DiffArmHome" AND ("r_S2_ArmZpos" = 0.0) AND ("r_S2_ArmXpos" = 0.0) AND "DO_S2_RotateLeft" AND "DO_S2_RotateRight";
   IF #_w1 THEN
       "DO_S2_RotateLeft" := FALSE;
       "DO_S2_RotateRight" := FALSE;
   END_IF;
END_REGION
END_FUNCTION

FUNCTION "Station3" : Void   // FC3, LAD
TITLE = Station 3 — Packaging & Palletizing
{ S7_Optimized_Access := 'TRUE' }
AUTHOR : Youness Tebbaq
VERSION : 0.1
// Station 3 (Packaging & Palletizing).
// -Final products are pushed into an elevator two at a time (Cnt_S3_ItemsInRow). 
// -After a 1-second debounce the pusher activates. The pallet is loaded with a row of items, the elevator raises to its upper limit, a clamp/plate sequence is executed (two	
// iterations), and the elevator lowers again. 
// -When a finished pallet reaches the exit sensor, the outfeed roller and remover start. The sequence uses three counters (counter_0 for items, counter_1 for the clamp/plate cycle, counter_2 for the elevator lower step) and three edge-trigger flags (b_S3_Trig_PalletLoaded, b_S3_Trig_OpenPlate, b_S3_Trig_PlateCycle).
   VAR_TEMP
      Tage_10 : Bool;
      rs_db : Bool;
   END_VAR
   VAR_TEMP   // added for the SCL form of the ladder/FBD networks
      _w1 : Bool;
      _w2 : Bool;
      _w3 : Bool;
      _w4 : Bool;
   END_VAR
BEGIN

REGION Network 1: Count items entering the row
   // Counter_0 (Cnt_S3_ItemsInRow, CTU instance) counts the parts
   // entering the station on the entry diffuse sensor (DI_S3_EntryPart). When
   // the count reaches 2 (PV=2), the counter's Q output goes high and triggers
   // the debounce timer in Network 2. The pusher limit sensor (DI_S3_PusherLimit)
   // resets the counter when the pusher retracts, so the next row can be counted.
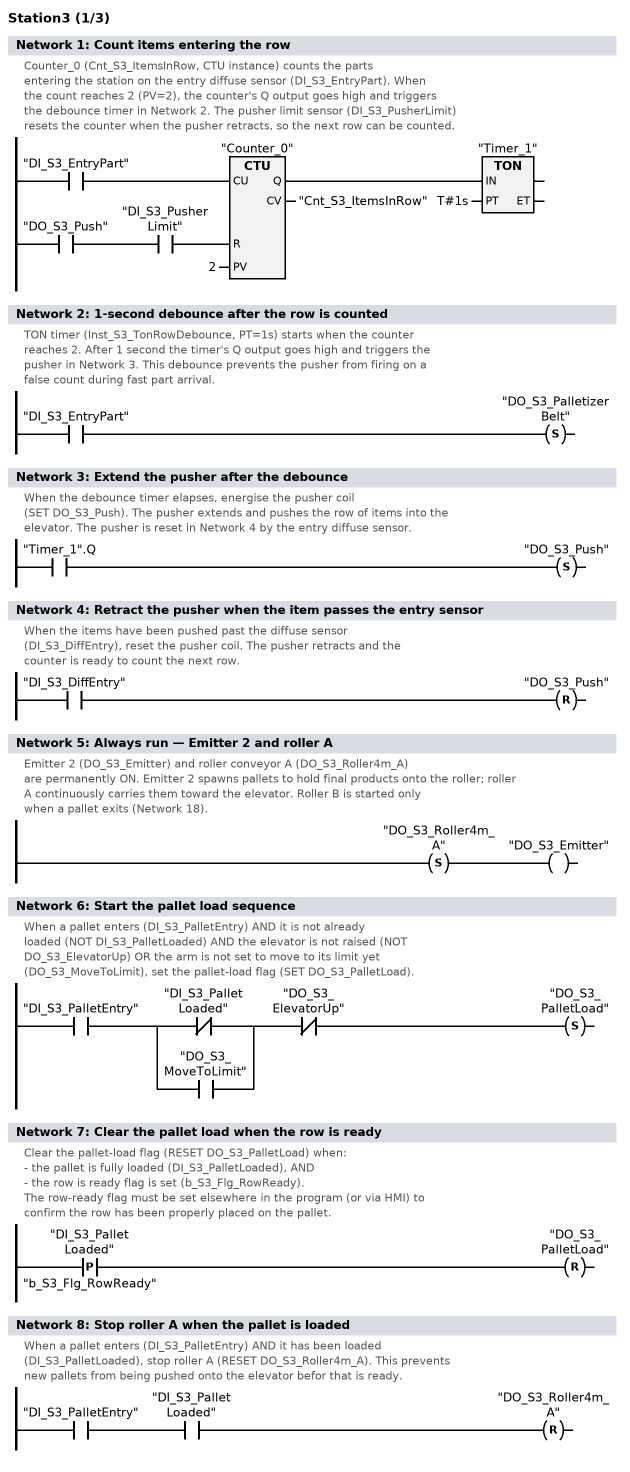
   "Counter_0".CTU(CU := "DI_S3_EntryPart",
                   R := "DO_S3_Push" AND "DI_S3_PusherLimit",
                   PV := 2,
                   CV => "Cnt_S3_ItemsInRow");
   "Timer_1".TON(IN := "Counter_0".Q, PT := T#1s);
END_REGION

REGION Network 2: 1-second debounce after the row is counted
   // TON timer (Inst_S3_TonRowDebounce, PT=1s) starts when the counter
   // reaches 2. After 1 second the timer's Q output goes high and triggers the
   // pusher in Network 3. This debounce prevents the pusher from firing on a
   // false count during fast part arrival.
   RUNG wire#powerrail
      Contact( "DI_S3_EntryPart" )
      S_Coil( "DO_S3_PalletizerBelt" )
   END_RUNG
   // the same network as SCL:
   IF "DI_S3_EntryPart" THEN "DO_S3_PalletizerBelt" := TRUE; END_IF;
END_REGION

REGION Network 3: Extend the pusher after the debounce
   // When the debounce timer elapses, energise the pusher coil
   // (SET DO_S3_Push). The pusher extends and pushes the row of items into the
   // elevator. The pusher is reset in Network 4 by the entry diffuse sensor.
   RUNG wire#powerrail
      Contact( "Timer_1".Q )
      S_Coil( "DO_S3_Push" )
   END_RUNG
   // the same network as SCL:
   IF "Timer_1".Q THEN "DO_S3_Push" := TRUE; END_IF;
END_REGION

REGION Network 4: Retract the pusher when the item passes the entry sensor
   // When the items have been pushed past the diffuse sensor
   // (DI_S3_DiffEntry), reset the pusher coil. The pusher retracts and the
   // counter is ready to count the next row.
   RUNG wire#powerrail
      Contact( "DI_S3_DiffEntry" )
      R_Coil( "DO_S3_Push" )
   END_RUNG
   // the same network as SCL:
   IF "DI_S3_DiffEntry" THEN "DO_S3_Push" := FALSE; END_IF;
END_REGION

REGION Network 5: Always run — Emitter 2 and roller A
   // Emitter 2 (DO_S3_Emitter) and roller conveyor A (DO_S3_Roller4m_A)
   // are permanently ON. Emitter 2 spawns pallets to hold final products onto the roller; roller
   // A continuously carries them toward the elevator. Roller B is started only
   // when a pallet exits (Network 18).
   RUNG wire#powerrail
      S_Coil( "DO_S3_Roller4m_A" )
      Coil( "DO_S3_Emitter" )
   END_RUNG
   // the same network as SCL:
   "DO_S3_Roller4m_A" := TRUE;
   "DO_S3_Emitter" := TRUE;
END_REGION

REGION Network 6: Start the pallet load sequence
   // When a pallet enters (DI_S3_PalletEntry) AND it is not already
   // loaded (NOT DI_S3_PalletLoaded) AND the elevator is not raised (NOT
   // DO_S3_ElevatorUp) OR the arm is not set to move to its limit yet
   // (DO_S3_MoveToLimit), set the pallet-load flag (SET DO_S3_PalletLoad).
   RUNG wire#powerrail
      Contact( "DI_S3_PalletEntry" )
      wire#w1
      I_Contact( "DI_S3_PalletLoaded" )
      wire#w2
      I_Contact( "DO_S3_ElevatorUp" )
      S_Coil( "DO_S3_PalletLoad" )
   END_RUNG
   RUNG wire#w1
      Contact( "DO_S3_MoveToLimit" )
   END_RUNG wire#w2
   // the same network as SCL:
   IF "DI_S3_PalletEntry" AND (NOT "DI_S3_PalletLoaded" OR "DO_S3_MoveToLimit") AND NOT "DO_S3_ElevatorUp" THEN
       "DO_S3_PalletLoad" := TRUE;
   END_IF;
END_REGION

REGION Network 7: Clear the pallet load when the row is ready
   // Clear the pallet-load flag (RESET DO_S3_PalletLoad) when:
   //   - the pallet is fully loaded (DI_S3_PalletLoaded), AND
   //   - the row is ready flag is set (b_S3_Flg_RowReady).
   // The row-ready flag must be set elsewhere in the program (or via HMI) to
   // confirm the row has been properly placed on the pallet.
   RUNG wire#powerrail
      P_Contact(operand := "DI_S3_PalletLoaded", bit := "b_S3_Flg_RowReady")
      R_Coil( "DO_S3_PalletLoad" )
   END_RUNG
   // the same network as SCL:
   #_w1 := "DI_S3_PalletLoaded" AND NOT "b_S3_Flg_RowReady";   // rising edge of "DI_S3_PalletLoaded"
   "b_S3_Flg_RowReady" := "DI_S3_PalletLoaded";
   IF #_w1 THEN "DO_S3_PalletLoad" := FALSE; END_IF;
END_REGION

REGION Network 8: Stop roller A when the pallet is loaded
   // When a pallet enters (DI_S3_PalletEntry) AND it has been loaded
   // (DI_S3_PalletLoaded), stop roller A (RESET DO_S3_Roller4m_A). This prevents
   // new pallets from being pushed onto the elevator befor that is ready.
   RUNG wire#powerrail
      Contact( "DI_S3_PalletEntry" )
      Contact( "DI_S3_PalletLoaded" )
      R_Coil( "DO_S3_Roller4m_A" )
   END_RUNG
   // the same network as SCL:
   IF "DI_S3_PalletEntry" AND "DI_S3_PalletLoaded" THEN "DO_S3_Roller4m_A" := FALSE; END_IF;
END_REGION

REGION Network 9: Start the elevator-up sequence on rising edge of pallet-loaded
   // On the rising edge of the pallet-loaded sensor (P_TRIG b_S3_Trig_PalletLoaded), energise BOTH the elevator-up coil (SET DO_S3_ElevatorUp) AND the move-to-limit coil (SET DO_S3_MoveToLimit).
   // The elevator starts raising and the arm drives to its upper position.
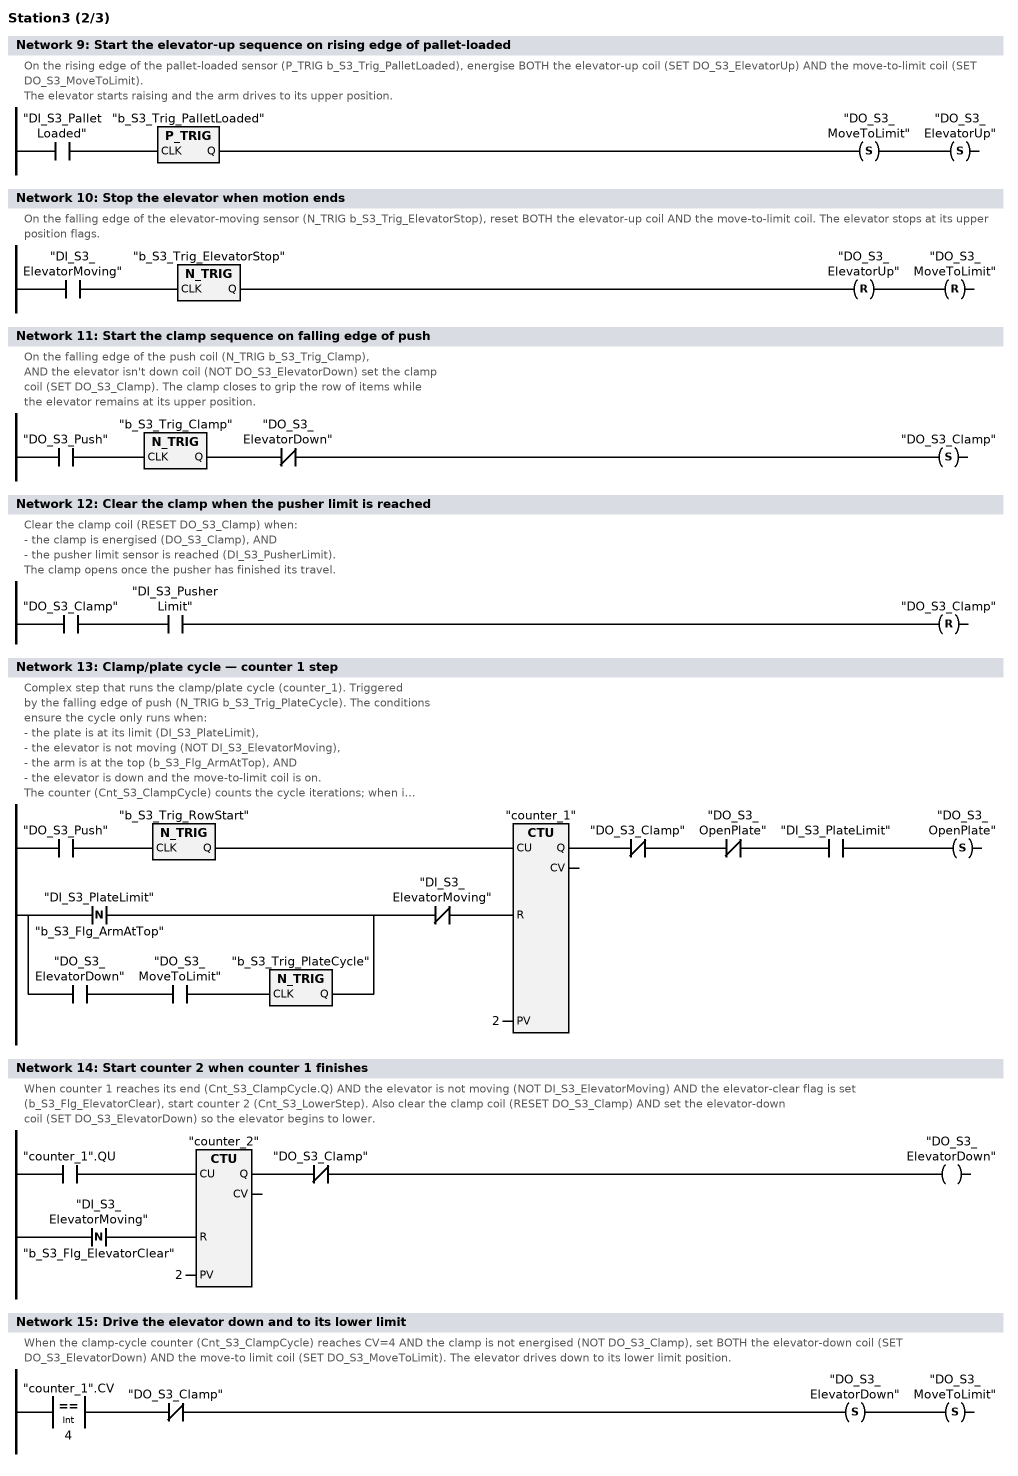
   RUNG wire#powerrail
      Contact( "DI_S3_PalletLoaded" )
      P_Trig( "b_S3_Trig_PalletLoaded" )
      S_Coil( "DO_S3_MoveToLimit" )
      S_Coil( "DO_S3_ElevatorUp" )
   END_RUNG
   // the same network as SCL:
   #_w1 := "DI_S3_PalletLoaded" AND NOT "b_S3_Trig_PalletLoaded";   // rising edge
   "b_S3_Trig_PalletLoaded" := "DI_S3_PalletLoaded";
   IF #_w1 THEN
       "DO_S3_MoveToLimit" := TRUE;
       "DO_S3_ElevatorUp" := TRUE;
   END_IF;
END_REGION

REGION Network 10: Stop the elevator when motion ends
   // On the falling edge of the elevator-moving sensor (N_TRIG b_S3_Trig_ElevatorStop), reset BOTH the elevator-up coil AND the move-to-limit coil. The elevator stops at its upper position flags.
   RUNG wire#powerrail
      Contact( "DI_S3_ElevatorMoving" )
      N_Trig( "b_S3_Trig_ElevatorStop" )
      R_Coil( "DO_S3_ElevatorUp" )
      R_Coil( "DO_S3_MoveToLimit" )
   END_RUNG
   // the same network as SCL:
   #_w1 := NOT "DI_S3_ElevatorMoving" AND "b_S3_Trig_ElevatorStop";   // falling edge
   "b_S3_Trig_ElevatorStop" := "DI_S3_ElevatorMoving";
   IF #_w1 THEN
       "DO_S3_ElevatorUp" := FALSE;
       "DO_S3_MoveToLimit" := FALSE;
   END_IF;
END_REGION

REGION Network 11: Start the clamp sequence on falling edge of push
   // On the falling edge of the push coil (N_TRIG b_S3_Trig_Clamp),
   // AND the elevator isn't down coil (NOT DO_S3_ElevatorDown) set the clamp
   // coil (SET DO_S3_Clamp). The clamp closes to grip the row of items while
   // the elevator remains at its upper position.
   RUNG wire#powerrail
      Contact( "DO_S3_Push" )
      N_Trig( "b_S3_Trig_Clamp" )
      I_Contact( "DO_S3_ElevatorDown" )
      S_Coil( "DO_S3_Clamp" )
   END_RUNG
   // the same network as SCL:
   #_w1 := NOT "DO_S3_Push" AND "b_S3_Trig_Clamp";   // falling edge
   "b_S3_Trig_Clamp" := "DO_S3_Push";
   IF #_w1 AND NOT "DO_S3_ElevatorDown" THEN "DO_S3_Clamp" := TRUE; END_IF;
END_REGION

REGION Network 12: Clear the clamp when the pusher limit is reached
   // Clear the clamp coil (RESET DO_S3_Clamp) when:
   //   - the clamp is energised (DO_S3_Clamp), AND
   //   - the pusher limit sensor is reached (DI_S3_PusherLimit).
   // The clamp opens once the pusher has finished its travel.
   RUNG wire#powerrail
      Contact( "DO_S3_Clamp" )
      Contact( "DI_S3_PusherLimit" )
      R_Coil( "DO_S3_Clamp" )
   END_RUNG
   // the same network as SCL:
   IF "DO_S3_Clamp" AND "DI_S3_PusherLimit" THEN "DO_S3_Clamp" := FALSE; END_IF;
END_REGION

REGION Network 13: Clamp/plate cycle — counter 1 step
   // Complex step that runs the clamp/plate cycle (counter_1). Triggered
   // by the falling edge of push (N_TRIG b_S3_Trig_PlateCycle). The conditions
   // ensure the cycle only runs when:
   //   - the plate is at its limit (DI_S3_PlateLimit),
   //   - the elevator is not moving (NOT DI_S3_ElevatorMoving),
   //   - the arm is at the top (b_S3_Flg_ArmAtTop), AND
   //   - the elevator is down and the move-to-limit coil is on.
   // The counter (Cnt_S3_ClampCycle) counts the cycle iterations; when it
   // reaches PV=2 the cycle ends. Then the clamp is reset, the open-plate flag
   // is reset, and the plate is opened (SET DO_S3_OpenPlate) when the plate
   // limit is no longer reached.
   #_w1 := NOT "DO_S3_Push" AND "b_S3_Trig_RowStart";   // falling edge
   "b_S3_Trig_RowStart" := "DO_S3_Push";
   #_w2 := NOT "DI_S3_PlateLimit" AND "b_S3_Flg_ArmAtTop";   // falling edge of "DI_S3_PlateLimit"
   "b_S3_Flg_ArmAtTop" := "DI_S3_PlateLimit";
   #_w3 := "DO_S3_ElevatorDown" AND "DO_S3_MoveToLimit";
   #_w4 := NOT #_w3 AND "b_S3_Trig_PlateCycle";   // falling edge
   "b_S3_Trig_PlateCycle" := #_w3;
   "counter_1".CTU(CU := #_w1, R := (#_w2 OR #_w4) AND NOT "DI_S3_ElevatorMoving", PV := 2);
   IF "counter_1".Q AND NOT "DO_S3_Clamp" AND NOT "DO_S3_OpenPlate" AND "DI_S3_PlateLimit" THEN
       "DO_S3_OpenPlate" := TRUE;
   END_IF;
END_REGION

REGION Network 14: Start counter 2 when counter 1 finishes
   // When counter 1 reaches its end (Cnt_S3_ClampCycle.Q) AND the elevator is not moving (NOT DI_S3_ElevatorMoving) AND the elevator-clear flag is set (b_S3_Flg_ElevatorClear), start counter 2 (Cnt_S3_LowerStep). Also clear the clamp coil (RESET DO_S3_Clamp) AND set the elevator-down
   // coil (SET DO_S3_ElevatorDown) so the elevator begins to lower.
   #_w1 := NOT "DI_S3_ElevatorMoving" AND "b_S3_Flg_ElevatorClear";   // falling edge of "DI_S3_ElevatorMoving"
   "b_S3_Flg_ElevatorClear" := "DI_S3_ElevatorMoving";
   "counter_2".CTU(CU := "counter_1".QU, R := #_w1, PV := 2);
   "DO_S3_ElevatorDown" := "counter_2".Q AND NOT "DO_S3_Clamp";
END_REGION

REGION Network 15: Drive the elevator down and to its lower limit
   // When the clamp-cycle counter (Cnt_S3_ClampCycle) reaches CV=4 AND the clamp is not energised (NOT DO_S3_Clamp), set BOTH the elevator-down coil (SET DO_S3_ElevatorDown) AND the move-to limit coil (SET DO_S3_MoveToLimit). The elevator drives down to its lower limit position.
   RUNG wire#powerrail
      { S7_Templates := "SrcType := Int" } EQ_Contact(in1 := "counter_1".CV, in2 := 4)
      I_Contact( "DO_S3_Clamp" )
      S_Coil( "DO_S3_ElevatorDown" )
      S_Coil( "DO_S3_MoveToLimit" )
   END_RUNG
   // the same network as SCL:
   IF ("counter_1".CV = 4) AND NOT "DO_S3_Clamp" THEN
       "DO_S3_ElevatorDown" := TRUE;
       "DO_S3_MoveToLimit" := TRUE;
   END_IF;
END_REGION

REGION Network 16: Open the plate when the elevator is fully down
   // When the elevator-down coil is energised (DO_S3_ElevatorDown) AND the falling edge of the open-plate trigger fires (N_TRIG b_S3_Trig_OpenPlate) AND the elevator-up coil is off (NOT DO_S3_ElevatorUp), increment counter 3 (Cnt_S3_PlateOpen) AND reset the open-plate coil (RESET DO_S3_OpenPlate). The plate is opened to release the loaded row onto the pallet.
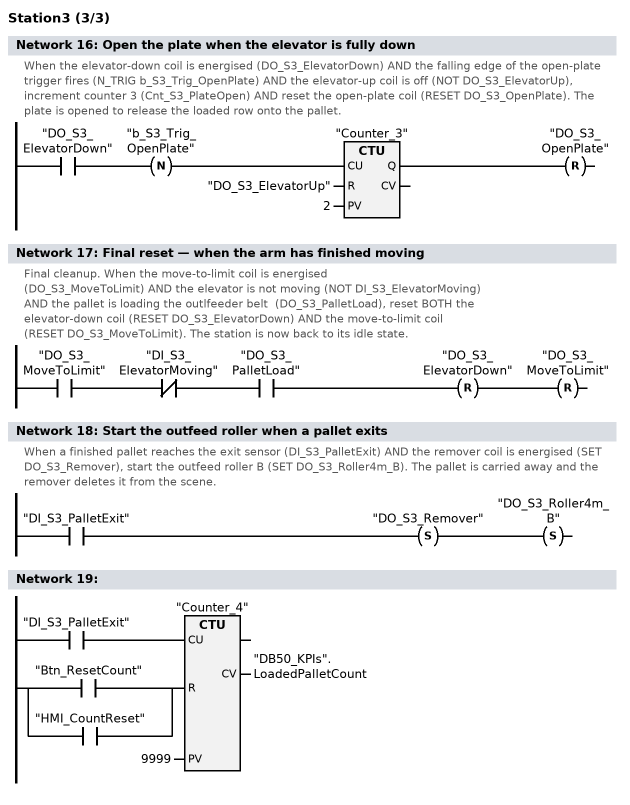
   #_w1 := NOT "DO_S3_ElevatorDown" AND "b_S3_Trig_OpenPlate";   // falling edge
   "b_S3_Trig_OpenPlate" := "DO_S3_ElevatorDown";
   "Counter_3".CTU(CU := #_w1, R := "DO_S3_ElevatorUp", PV := 2);
   IF "Counter_3".Q THEN "DO_S3_OpenPlate" := FALSE; END_IF;
END_REGION

REGION Network 17: Final reset — when the arm has finished moving
   // Final cleanup. When the move-to-limit coil is energised
   // (DO_S3_MoveToLimit) AND the elevator is not moving (NOT DI_S3_ElevatorMoving)
   // AND the pallet is loading the outlfeeder belt  (DO_S3_PalletLoad), reset BOTH the
   // elevator-down coil (RESET DO_S3_ElevatorDown) AND the move-to-limit coil
   // (RESET DO_S3_MoveToLimit). The station is now back to its idle state.
   RUNG wire#powerrail
      Contact( "DO_S3_MoveToLimit" )
      I_Contact( "DI_S3_ElevatorMoving" )
      Contact( "DO_S3_PalletLoad" )
      R_Coil( "DO_S3_ElevatorDown" )
      R_Coil( "DO_S3_MoveToLimit" )
   END_RUNG
   // the same network as SCL:
   IF "DO_S3_MoveToLimit" AND NOT "DI_S3_ElevatorMoving" AND "DO_S3_PalletLoad" THEN
       "DO_S3_ElevatorDown" := FALSE;
       "DO_S3_MoveToLimit" := FALSE;
   END_IF;
END_REGION

REGION Network 18: Start the outfeed roller when a pallet exits
   // When a finished pallet reaches the exit sensor (DI_S3_PalletExit) AND the remover coil is energised (SET DO_S3_Remover), start the outfeed roller B (SET DO_S3_Roller4m_B). The pallet is carried away and the remover deletes it from the scene.
   RUNG wire#powerrail
      Contact( "DI_S3_PalletExit" )
      S_Coil( "DO_S3_Remover" )
      S_Coil( "DO_S3_Roller4m_B" )
   END_RUNG
   // the same network as SCL:
   IF "DI_S3_PalletExit" THEN
       "DO_S3_Remover" := TRUE;
       "DO_S3_Roller4m_B" := TRUE;
   END_IF;
END_REGION

REGION Network 19
   "Counter_4".CTU(CU := "DI_S3_PalletExit",
                   R := "Btn_ResetCount" OR "HMI_CountReset",
                   PV := 9999,
                   CV => "DB50_KPIs".LoadedPalletCount);
END_REGION
END_FUNCTION

FUNCTION "ControlPanel" : Void   // FC4, LAD
{ S7_Optimized_Access := 'TRUE' }
VERSION : 0.1
   VAR_TEMP   // added for the SCL form of the ladder/FBD networks
      _w1 : Bool;
   END_VAR
BEGIN

REGION Network 1
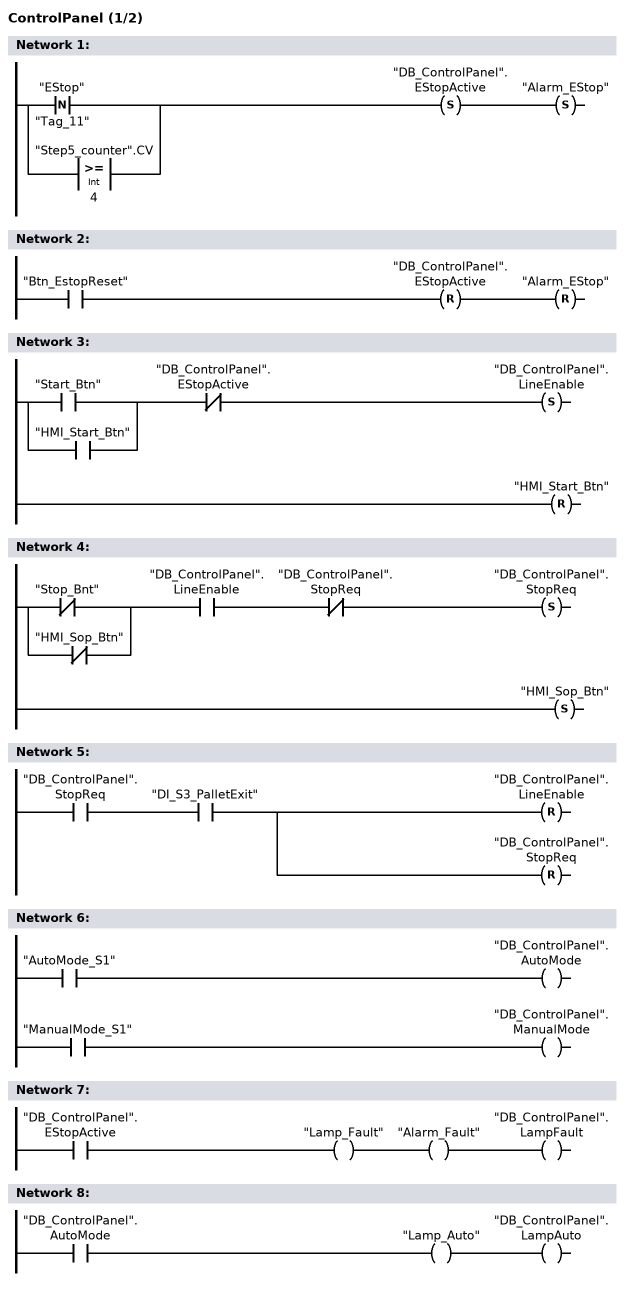
   RUNG wire#powerrail
      N_Contact(operand := "EStop", bit := "Tag_11")
      wire#w1
      S_Coil( "DB_ControlPanel".EStopActive )
      S_Coil( "Alarm_EStop" )
   END_RUNG
   RUNG wire#powerrail
      { S7_Templates := "SrcType := Int" } GE_Contact(in1 := "Step5_counter".CV, in2 := 4)
   END_RUNG wire#w1
   // the same network as SCL:
   #_w1 := NOT "EStop" AND "Tag_11";   // falling edge of "EStop"
   "Tag_11" := "EStop";
   IF #_w1 OR ("Step5_counter".CV >= 4) THEN
       "DB_ControlPanel".EStopActive := TRUE;
       "Alarm_EStop" := TRUE;
   END_IF;
END_REGION

REGION Network 2
   RUNG wire#powerrail
      Contact( "Btn_EstopReset" )
      R_Coil( "DB_ControlPanel".EStopActive )
      R_Coil( "Alarm_EStop" )
   END_RUNG
   // the same network as SCL:
   IF "Btn_EstopReset" THEN
       "DB_ControlPanel".EStopActive := FALSE;
       "Alarm_EStop" := FALSE;
   END_IF;
END_REGION

REGION Network 3
   RUNG wire#powerrail
      Contact( "Start_Btn" )
      wire#w1
      I_Contact( "DB_ControlPanel".EStopActive )
      S_Coil( "DB_ControlPanel".LineEnable )
   END_RUNG
   RUNG wire#powerrail
      Contact( "HMI_Start_Btn" )
   END_RUNG wire#w1
   RUNG wire#powerrail
      R_Coil( "HMI_Start_Btn" )
   END_RUNG
   // the same network as SCL:
   IF ("Start_Btn" OR "HMI_Start_Btn") AND NOT "DB_ControlPanel".EStopActive THEN
       "DB_ControlPanel".LineEnable := TRUE;
   END_IF;
   "HMI_Start_Btn" := FALSE;
END_REGION

REGION Network 4
   RUNG wire#powerrail
      I_Contact( "Stop_Bnt" )
      wire#w1
      Contact( "DB_ControlPanel".LineEnable )
      I_Contact( "DB_ControlPanel".StopReq )
      S_Coil( "DB_ControlPanel".StopReq )
   END_RUNG
   RUNG wire#powerrail
      I_Contact( "HMI_Sop_Btn" )
   END_RUNG wire#w1
   RUNG wire#powerrail
      S_Coil( "HMI_Sop_Btn" )
   END_RUNG
   // the same network as SCL:
   IF (NOT "Stop_Bnt" OR NOT "HMI_Sop_Btn") AND "DB_ControlPanel".LineEnable AND NOT "DB_ControlPanel".StopReq THEN
       "DB_ControlPanel".StopReq := TRUE;
   END_IF;
   "HMI_Sop_Btn" := TRUE;
END_REGION

REGION Network 5
   RUNG wire#powerrail
      Contact( "DB_ControlPanel".StopReq )
      Contact( "DI_S3_PalletExit" )
      wire#w1
      R_Coil( "DB_ControlPanel".LineEnable )
   END_RUNG
   RUNG wire#w1
      R_Coil( "DB_ControlPanel".StopReq )
   END_RUNG
   // the same network as SCL:
   IF "DB_ControlPanel".StopReq AND "DI_S3_PalletExit" THEN
       "DB_ControlPanel".LineEnable := FALSE;
       "DB_ControlPanel".StopReq := FALSE;
   END_IF;
END_REGION

REGION Network 6
   RUNG wire#powerrail
      Contact( "AutoMode_S1" )
      Coil( "DB_ControlPanel".AutoMode )
   END_RUNG
   RUNG wire#powerrail
      Contact( "ManualMode_S1" )
      Coil( "DB_ControlPanel".ManualMode )
   END_RUNG
   // the same network as SCL:
   "DB_ControlPanel".AutoMode := "AutoMode_S1";
   "DB_ControlPanel".ManualMode := "ManualMode_S1";
END_REGION

REGION Network 7
   RUNG wire#powerrail
      Contact( "DB_ControlPanel".EStopActive )
      Coil( "Lamp_Fault" )
      Coil( "Alarm_Fault" )
      Coil( "DB_ControlPanel".LampFault )
   END_RUNG
   // the same network as SCL:
   "Lamp_Fault" := "DB_ControlPanel".EStopActive;
   "Alarm_Fault" := "DB_ControlPanel".EStopActive;
   "DB_ControlPanel".LampFault := "DB_ControlPanel".EStopActive;
END_REGION

REGION Network 8
   RUNG wire#powerrail
      Contact( "DB_ControlPanel".AutoMode )
      Coil( "Lamp_Auto" )
      Coil( "DB_ControlPanel".LampAuto )
   END_RUNG
   // the same network as SCL:
   "Lamp_Auto" := "DB_ControlPanel".AutoMode;
   "DB_ControlPanel".LampAuto := "DB_ControlPanel".AutoMode;
END_REGION

REGION Network 9
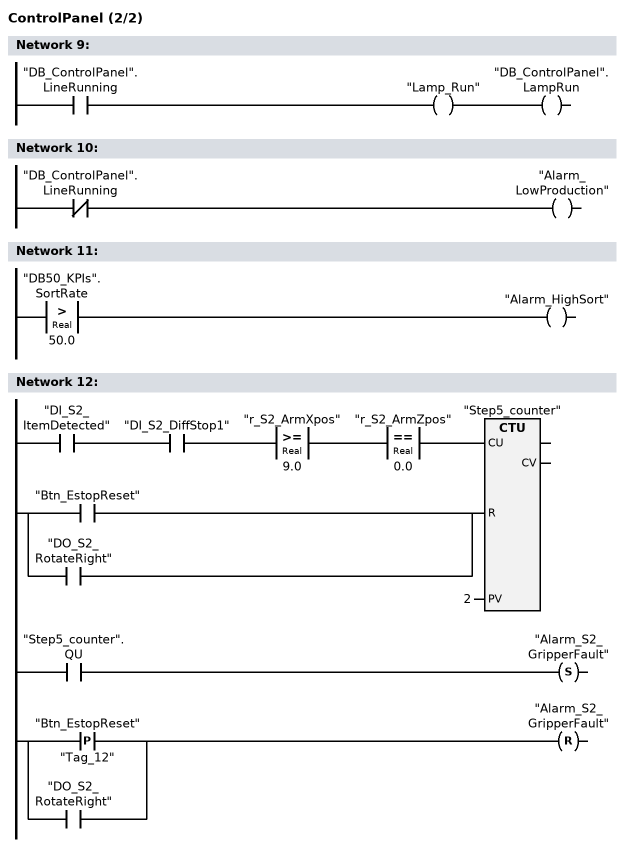
   RUNG wire#powerrail
      Contact( "DB_ControlPanel".LineRunning )
      Coil( "Lamp_Run" )
      Coil( "DB_ControlPanel".LampRun )
   END_RUNG
   // the same network as SCL:
   "Lamp_Run" := "DB_ControlPanel".LineRunning;
   "DB_ControlPanel".LampRun := "DB_ControlPanel".LineRunning;
END_REGION

REGION Network 10
   RUNG wire#powerrail
      I_Contact( "DB_ControlPanel".LineRunning )
      Coil( "Alarm_LowProduction" )
   END_RUNG
   // the same network as SCL:
   "Alarm_LowProduction" := NOT "DB_ControlPanel".LineRunning;
END_REGION

REGION Network 11
   RUNG wire#powerrail
      { S7_Templates := "SrcType := Real" } GT_Contact(in1 := "DB50_KPIs".SortRate, in2 := 50.0)
      Coil( "Alarm_HighSort" )
   END_RUNG
   // the same network as SCL:
   "Alarm_HighSort" := "DB50_KPIs".SortRate > 50.0;
END_REGION

REGION Network 12
   "Step5_counter".CTU(CU := "DI_S2_ItemDetected" AND "DI_S2_DiffStop1" AND ("r_S2_ArmXpos" >= 9.0) AND ("r_S2_ArmZpos" = 0.0),
                       R := "Btn_EstopReset" OR "DO_S2_RotateRight",
                       PV := 2);
   IF "Step5_counter".QU THEN "Alarm_S2_GripperFault" := TRUE; END_IF;
   #_w1 := "Btn_EstopReset" AND NOT "Tag_12";   // rising edge of "Btn_EstopReset"
   "Tag_12" := "Btn_EstopReset";
   IF #_w1 OR "DO_S2_RotateRight" THEN "Alarm_S2_GripperFault" := FALSE; END_IF;
END_REGION
END_FUNCTION

ORGANIZATION_BLOCK "Main"   // OB1, LAD, ProgramCycle
TITLE = "SmartLine 360 — Main Program Sweep"
{ S7_Optimized_Access := 'TRUE' }
AUTHOR : Youness Tebbaq
VERSION : 0.1
// "Main program sweep. Calls the lab function only in the first cycle, then runs the three stations in sequence: Station 1 (Infeed & Color Sorting) → Station 2 (Assembly) → Station 3 (Packaging & Palletizing). Every station is a Function Call (FC) so that each one can be compiled and tested independently."
   VAR_INPUT
      Initial_Call : Bool;   // Initial call of this OB
      Remanence : Bool;   // =True, if remanent data are available
   END_VAR
   VAR_TEMP   // added for the SCL form of the ladder/FBD networks
      _w1 : Bool;
   END_VAR
BEGIN

REGION Network 1: S1 pusher extend coil
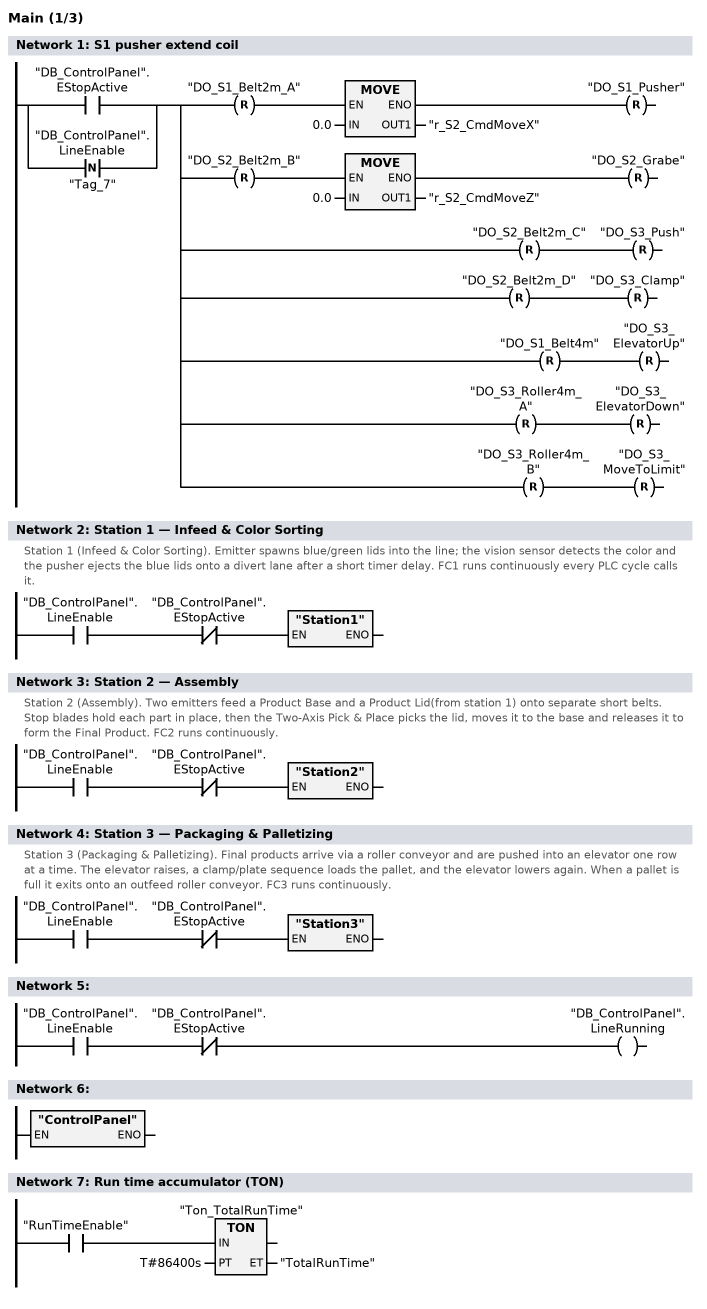
   RUNG wire#powerrail
      Contact( "DB_ControlPanel".EStopActive )
      wire#w1
      R_Coil( "DO_S1_Belt2m_A" )
      Move(in := 0.0, out1 => "r_S2_CmdMoveX")
      R_Coil( "DO_S1_Pusher" )
   END_RUNG
   RUNG wire#powerrail
      N_Contact(operand := "DB_ControlPanel".LineEnable, bit := "Tag_7")
   END_RUNG wire#w1
   RUNG wire#w1
      R_Coil( "DO_S2_Belt2m_B" )
      Move(in := 0.0, out1 => "r_S2_CmdMoveZ")
      R_Coil( "DO_S2_Grabe" )
   END_RUNG
   RUNG wire#w1
      R_Coil( "DO_S2_Belt2m_C" )
      R_Coil( "DO_S3_Push" )
   END_RUNG
   RUNG wire#w1
      R_Coil( "DO_S2_Belt2m_D" )
      R_Coil( "DO_S3_Clamp" )
   END_RUNG
   RUNG wire#w1
      R_Coil( "DO_S1_Belt4m" )
      R_Coil( "DO_S3_ElevatorUp" )
   END_RUNG
   RUNG wire#w1
      R_Coil( "DO_S3_Roller4m_A" )
      R_Coil( "DO_S3_ElevatorDown" )
   END_RUNG
   RUNG wire#w1
      R_Coil( "DO_S3_Roller4m_B" )
      R_Coil( "DO_S3_MoveToLimit" )
   END_RUNG
   // the same network as SCL:
   #_w1 := NOT "DB_ControlPanel".LineEnable AND "Tag_7";   // falling edge of "DB_ControlPanel".LineEnable
   "Tag_7" := "DB_ControlPanel".LineEnable;
   IF "DB_ControlPanel".EStopActive OR #_w1 THEN
       "DO_S1_Belt2m_A" := FALSE;
       "r_S2_CmdMoveX" := 0.0;
       "DO_S1_Pusher" := FALSE;
       "DO_S2_Belt2m_B" := FALSE;
       "r_S2_CmdMoveZ" := 0.0;
       "DO_S2_Grabe" := FALSE;
       "DO_S2_Belt2m_C" := FALSE;
       "DO_S3_Push" := FALSE;
       "DO_S2_Belt2m_D" := FALSE;
       "DO_S3_Clamp" := FALSE;
       "DO_S1_Belt4m" := FALSE;
       "DO_S3_ElevatorUp" := FALSE;
       "DO_S3_Roller4m_A" := FALSE;
       "DO_S3_ElevatorDown" := FALSE;
       "DO_S3_Roller4m_B" := FALSE;
       "DO_S3_MoveToLimit" := FALSE;
   END_IF;
END_REGION

REGION Network 2: Station 1 — Infeed & Color Sorting
   // Station 1 (Infeed & Color Sorting). Emitter spawns blue/green lids into the line; the vision sensor detects the color and the pusher ejects the blue lids onto a divert lane after a short timer delay. FC1 runs continuously every PLC cycle calls it.
   RUNG wire#powerrail
      Contact( "DB_ControlPanel".LineEnable )
      I_Contact( "DB_ControlPanel".EStopActive )
      "Station1"()
   END_RUNG
   // the same network as SCL:
   IF "DB_ControlPanel".LineEnable AND NOT "DB_ControlPanel".EStopActive THEN "Station1"(); END_IF;
END_REGION

REGION Network 3: Station 2 — Assembly
   // Station 2 (Assembly). Two emitters feed a Product Base and a Product Lid(from station 1) onto separate short belts. Stop blades hold each part in place, then the Two-Axis Pick & Place picks the lid, moves it to the base and releases it to form the Final Product. FC2 runs continuously.
   RUNG wire#powerrail
      Contact( "DB_ControlPanel".LineEnable )
      I_Contact( "DB_ControlPanel".EStopActive )
      "Station2"()
   END_RUNG
   // the same network as SCL:
   IF "DB_ControlPanel".LineEnable AND NOT "DB_ControlPanel".EStopActive THEN "Station2"(); END_IF;
END_REGION

REGION Network 4: Station 3 — Packaging & Palletizing
   // Station 3 (Packaging & Palletizing). Final products arrive via a roller conveyor and are pushed into an elevator one row at a time. The elevator raises, a clamp/plate sequence loads the pallet, and the elevator lowers again. When a pallet is full it exits onto an outfeed roller conveyor. FC3 runs continuously.
   RUNG wire#powerrail
      Contact( "DB_ControlPanel".LineEnable )
      I_Contact( "DB_ControlPanel".EStopActive )
      "Station3"()
   END_RUNG
   // the same network as SCL:
   IF "DB_ControlPanel".LineEnable AND NOT "DB_ControlPanel".EStopActive THEN "Station3"(); END_IF;
END_REGION

REGION Network 5
   RUNG wire#powerrail
      Contact( "DB_ControlPanel".LineEnable )
      I_Contact( "DB_ControlPanel".EStopActive )
      Coil( "DB_ControlPanel".LineRunning )
   END_RUNG
   // the same network as SCL:
   "DB_ControlPanel".LineRunning := "DB_ControlPanel".LineEnable AND NOT "DB_ControlPanel".EStopActive;
END_REGION

REGION Network 6
   RUNG wire#powerrail
      "ControlPanel"()
   END_RUNG
   // the same network as SCL:
   "ControlPanel"();
END_REGION

REGION Network 7: Run time accumulator (TON)
   "Ton_TotalRunTime".TON(IN := "RunTimeEnable", PT := T#86400s, ET => "TotalRunTime");
END_REGION

REGION Network 8: Down time accumulator (TON)
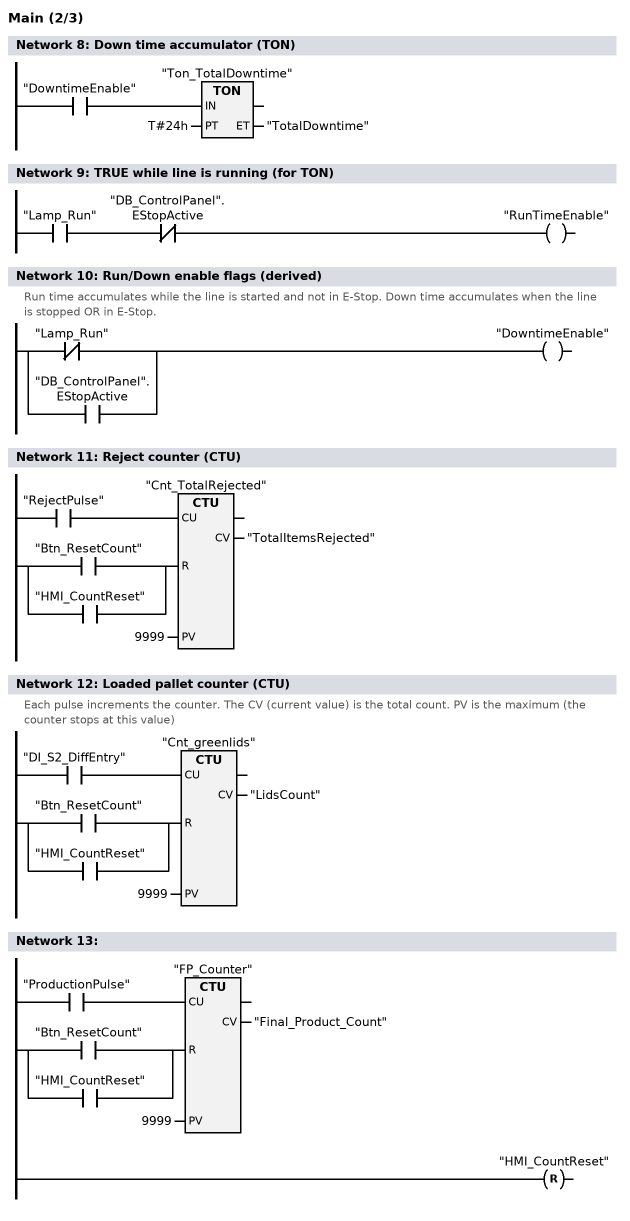
   "Ton_TotalDowntime".TON(IN := "DowntimeEnable", PT := T#24h, ET => "TotalDowntime");
END_REGION

REGION Network 9: TRUE while line is running (for TON)
   RUNG wire#powerrail
      Contact( "Lamp_Run" )
      I_Contact( "DB_ControlPanel".EStopActive )
      Coil( "RunTimeEnable" )
   END_RUNG
   // the same network as SCL:
   "RunTimeEnable" := "Lamp_Run" AND NOT "DB_ControlPanel".EStopActive;
END_REGION

REGION Network 10: Run/Down enable flags (derived)
   // Run time accumulates while the line is started and not in E-Stop. Down time accumulates when the line is stopped OR in E-Stop.
   RUNG wire#powerrail
      I_Contact( "Lamp_Run" )
      wire#w1
      Coil( "DowntimeEnable" )
   END_RUNG
   RUNG wire#powerrail
      Contact( "DB_ControlPanel".EStopActive )
   END_RUNG wire#w1
   // the same network as SCL:
   "DowntimeEnable" := NOT "Lamp_Run" OR "DB_ControlPanel".EStopActive;
END_REGION

REGION Network 11: Reject counter (CTU)
   "Cnt_TotalRejected".CTU(CU := "RejectPulse",
                           R := "Btn_ResetCount" OR "HMI_CountReset",
                           PV := 9999,
                           CV => "TotalItemsRejected");
END_REGION

REGION Network 12: Loaded pallet counter (CTU)
   // Each pulse increments the counter. The CV (current value) is the total count. PV is the maximum (the counter stops at this value)
   "Cnt_greenlids".CTU(CU := "DI_S2_DiffEntry",
                       R := "Btn_ResetCount" OR "HMI_CountReset",
                       PV := 9999,
                       CV => "LidsCount");
END_REGION

REGION Network 13
   "FP_Counter".CTU(CU := "ProductionPulse",
                    R := "Btn_ResetCount" OR "HMI_CountReset",
                    PV := 9999,
                    CV => "Final_Product_Count");
   "HMI_CountReset" := FALSE;
END_REGION

REGION Network 14
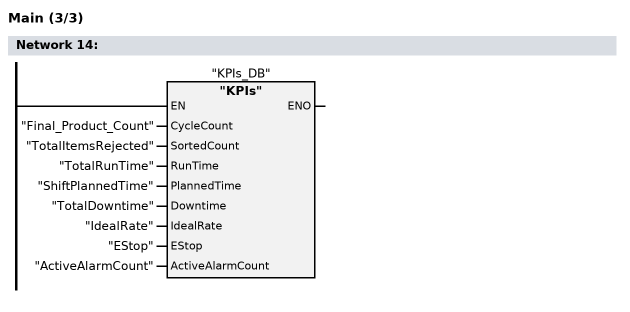
   RUNG wire#powerrail
      "KPIs_DB"(CycleCount := "Final_Product_Count", SortedCount := "TotalItemsRejected", RunTime := "TotalRunTime", PlannedTime := "ShiftPlannedTime", Downtime := "TotalDowntime", IdealRate := "IdealRate", ActiveAlarmCount := "ActiveAlarmCount", EStop := "EStop")
   END_RUNG
   // the same network as SCL:
   "KPIs_DB"(CycleCount := "Final_Product_Count",   // "KPIs"
             SortedCount := "TotalItemsRejected",
             RunTime := "TotalRunTime",
             PlannedTime := "ShiftPlannedTime",
             Downtime := "TotalDowntime",
             IdealRate := "IdealRate",
             EStop := "EStop",
             ActiveAlarmCount := "ActiveAlarmCount");
END_REGION
END_ORGANIZATION_BLOCK

ORGANIZATION_BLOCK "Startup"   // OB100, LAD, Startup
TITLE = "Complete Restart"
{ S7_Optimized_Access := 'TRUE' }
VERSION : 0.1
   VAR_INPUT
      LostRetentive : Bool;   // True if retentive data are lost
      LostRTC : Bool;   // True if date and time are lost
   END_VAR
BEGIN

REGION Network 1
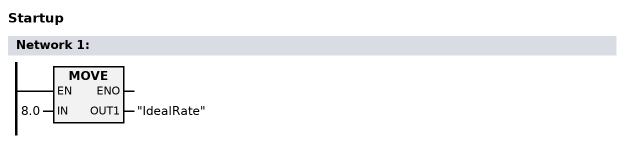
   RUNG wire#powerrail
      Move(in := 8.0, out1 => "IdealRate")
   END_RUNG
   // the same network as SCL:
   "IdealRate" := 8.0;
END_REGION
END_ORGANIZATION_BLOCK